(* CODESYS project Templates.export

Project tree, tasks and I/O mapping:
  Templates/
    Behaviour Model/
      function block ETrigATlTo_Temp [ST]: CleanupAction, CyclicAction, ExitAction, ResetAction, SampleAction, StartAction
      function block ETrigATl_Temp [ST]: CleanupAction, CyclicAction, ExitAction, ResetAction, SampleAction, StartAction
      function block ETrigATo_Temp [ST]: CleanupAction, CyclicAction, ExitAction, ResetAction, SampleAction, StartAction
      function block ETrigA_Temp [ST]: CleanupAction, CyclicAction, ExitAction, ResetAction, SampleAction, StartAction
      function block ETrigTlTo_Temp [ST]: CleanupAction, CyclicAction, ExitAction, ResetAction, SampleAction, StartAction
      function block ETrigTl_Temp [ST]: CleanupAction, CyclicAction, ExitAction, ResetAction, SampleAction, StartAction
      function block ETrigTo_Temp [ST]: CleanupAction, CyclicAction, ExitAction, ResetAction, SampleAction, StartAction
      function block ETrig_Temp [ST]: CleanupAction, CyclicAction, ExitAction, ResetAction, SampleAction, StartAction
      function block LConC_Temp [ST]: CleanupAction, CyclicAction, ExitAction, ResetAction, StartAction
      function block LConTlC_Temp [ST]: CleanupAction, CyclicAction, ExitAction, ResetAction, StartAction
      function block LConTlTo_Temp [ST]: CleanupAction, CyclicAction, ExitAction, ResetAction, StartAction
      function block LConTl_Temp [ST]: CleanupAction, CyclicAction, ExitAction, ResetAction, StartAction
      function block LConTo_Temp [ST]: CleanupAction, CyclicAction, ExitAction, ResetAction, StartAction
      function block LCon_Temp [ST]: CleanupAction, CyclicAction, ExitAction, ResetAction, StartAction
    FB Factory/
      function block CustomData [ST]
      function block CustomFB [ST]: prvInstInit
      function block CustomFBFactory_heap [ST]: Create, prvInstCount, prvInstPoolExtendsFactor, prvInstSize
      function block CustomFBFactory_static [ST]: Create, prvInstPoolAdr, prvInstPoolSize, prvInstSize
*)

// Templates/Behaviour Model/ETrigATlTo_Temp
//{attribute 'hide_all_locals'}
//{attribute 'conditionalshow_all_locals' := 'SomeText'}
//{attribute 'conditionalshow_all_locals'}
//{attribute 'conditionalshow' := 'SomeText'}
//{attribute 'conditionalshow'}
//{attribute 'hide'}
FUNCTION_BLOCK ETrigATlTo_Temp EXTENDS CBML.ETrigATlTo
VAR_INPUT
	(* specific Inputs *)
END_VAR
VAR_OUTPUT
	(* specific Outputs *)
	eErrorID : ERROR;
END_VAR
VAR
	(* specific vars *)
END_VAR

SUPER^();
IF _Model.iErrorID = CBML.ERROR.TIME_OUT THEN
	eErrorID := ERROR.TIME_OUT;
ELSE
	eErrorID := _Model.iErrorID;
END_IF

METHOD CleanupAction
VAR_INPUT
    xAbortProposed : BOOL;
    iErrorIDProposed: INT;
END_VAR
VAR_OUTPUT
    xComplete : BOOL := TRUE;
    xAbort: BOOL := xAbortProposed;
 	iErrorID : INT := iErrorIDProposed;
END_VAR
{analysis -2} 
/// ``CleanupAction`` is running until one of the following events occurs:
/// When ``xComplete`` is ``TRUE`` the state |STATE.DONE| is reached.
/// When ``xAbort`` is ``TRUE`` the state |STATE.ABORTED| is reached.
/// When ``iErrorID`` ≠ 0 (Zero) the state |STATE.ERROR| is reached.
///
/// | After a *Ready Condition* as input (``iErrorIDProposed`` = 0 and ``xAbortProposed`` = ``FALSE``), only the output states
/// | `DONE` (``xComplete`` is ``TRUE``) or `ERROR` (``iErrorID`` ≠ 0) are possible.
///
/// | After a *Error Condition* as input (``iErrorIDProposed`` ≠ 0), only the output state
/// | `ERROR` (``iErrorID`` ≠ 0) is possible.
///
/// | After a *Abort Condition* as Input (``xAbortProposed`` = ``TRUE``), only the output states
/// | `ABORTED` (``xAbort`` is ``TRUE``) or `ERROR` (``iErrorID`` ≠ 0) are possible.
///
/// .. admonition:: Example
///
///     .. code-block:: codesys
///     
///         (* common cleanup -- first steps *) 
///         
///         IF xComplete THEN
///             IF xAbortProposed THEN
///                 (* abort condition -- abort specific cleanup *)
///                 xAbort := TRUE;
///                 xComplete := FALSE;
///             ELSIF iErrorIDProposed <> 0 THEN
///                 (* error condition -- error specific cleanup *)
///                 iErrorID := SEL(xComplete, 0, iErrorIDProposed);
///                 xComplete := FALSE;
///             ELSE
///                 (* ready condition -- done specific cleanup*)
///             END_IF
///         END_IF
///
///         (* common cleanup -- last steps *) 
///
/// .. note::
///
///    If this method will not provide any implementation, please remove it!
END_METHOD

METHOD CyclicAction
VAR_INPUT
    itfTimingController : CBML.ITimingController;
END_VAR
VAR_OUTPUT
    xComplete : BOOL := TRUE;
    iErrorID : INT := 0;
END_VAR
{analysis -2} 
/// The CyclicAction is running until either ``xComplete`` is ``TRUE`` or ``iErrorID`` ≠  0 (Zero).
/// If ``xComplete`` is ``TRUE`` or ``iErrorID`` ≠  0 (Zero) the state |STATE.CLEANING| is reached.
/// With ``itfTimingController`` ≠  0 (Zero) it is possible to check the current invocation time (see: |ITimingController.ControllerCheckTiming|).
/// Function blocks with a ``udiTimeLimit`` input variable (see: |IETrigTl|, |IETrigATl|, |IETrigTlTo|, |IETrigATlTo|, |ILConTl|, |ILConTlTo|, |ILConTlC|)
/// should be implement in such a way that the current invocation is exited when the consumed time for this invocation has exceeded the settings from udiTimeLimit.
///
/// .. admonition:: Example
///
///     .. code-block:: codesys
///     
///         REPEAT
///             // working to reach the ready condition
///             // ⇒ xComplete := TRUE
///             // if the maximum invocation time is reached
///             // ⇒ xTimeLimit := TRUE
///             // if the maximum operating time is reached
///             // ⇒ xTimeOut := TRUE
///             // if an error condition is reached
///             // ⇒ set iErrorID to a value other than 0 (Zero)
///             itfTimingController.ControllerCheckTiming(
///                 xTimeOut=>xTimeOut,
///                 xTimeLimit=>xTimeLimit
///             );
///         
///             xComplete := TRUE;
///             iErrorID := ERROR.NO_ERROR;
///     
///         UNTIL xComplete OR
///               xTimeOut OR xTimeLimit OR
///               iErrorID <> ERROR.NO_ERROR
///         END_REPEAT
///
/// .. note::
///
///    If this method will not provide any implementation, please remove it!
END_METHOD

METHOD ExitAction
VAR_INPUT
    xAfterCleanup : BOOL;
    xInCopyCode : BOOL;
END_VAR
{analysis -2} 
/// This method is intended for releasing external resources (like RTS handles).
/// Do not call other internal function block instances in the context of this method.
/// Call only external functions defined inside the RTS.
/// For cleaning up other resources then external ones, please use the ``CleanupAction``.
/// This method should be callable in the context of ``FB_EXIT`` for example
/// before downloading a new application or before reseting an application.
///
/// .. note::
///
///    If this method will not provide any implementation, please remove it!
END_METHOD

METHOD ResetAction
VAR_OUTPUT
    xComplete : BOOL := TRUE;
END_VAR
{analysis -2} 
/// The ``ResetAction`` is running until the output ``xComplete`` is ``TRUE``.
/// If ``xComplete`` is ``TRUE`` the state |STATE.DORMANT| is reached.
///
/// .. note::
///
///    If this method will not provide any implementation, please remove it!
END_METHOD

METHOD SampleAction
VAR_OUTPUT
 	iErrorID : INT := 0;
END_VAR
{analysis -2} 
/// After leaving the state |STATE.DORMANT| the ``SampleAction`` is running one time then the state |STATE.STARTING| is reached.
/// If there is a ``iErrorID`` ≠  0 (Zero) the state |STATE.CLEANING| is reached instead.
///
/// .. note::
///
///    If this method will not provide any implementation, please remove it!
END_METHOD

METHOD StartAction
VAR_OUTPUT
    xComplete : BOOL := TRUE;
	iErrorID : INT := 0;
END_VAR
{analysis -2} 
/// The ``StartAction`` is running until either the output ``xComplete`` is ``TRUE`` or ``iErrorID`` ≠ 0 (Zero).
/// If ``xComplete`` is ``TRUE`` the state |STATE.EXECUTING| is reached.
/// If there is a ``iErrorID`` ≠  0 (Zero) the state |STATE.CLEANING| is reached.
///
/// .. note::
///
///    To sample the inputs in the first invocation of a function block the method SampleAction is the solution of choice.
///    See: |ISampleActionProvider.SampleAction|
///
/// .. note::
///
///    If this method will not provide any implementation, please remove it!
END_METHOD

END_FUNCTION_BLOCK

// Templates/Behaviour Model/ETrigATl_Temp
//{attribute 'hide_all_locals'}
//{attribute 'conditionalshow_all_locals' := 'SomeText'}
//{attribute 'conditionalshow_all_locals'}
//{attribute 'conditionalshow' := 'SomeText'}
//{attribute 'conditionalshow'}
//{attribute 'hide'}
FUNCTION_BLOCK ETrigATl_Temp EXTENDS CBML.ETrigATl
VAR_INPUT
	(* specific Inputs *)
END_VAR
VAR_OUTPUT
	eErrorID : ERROR;
	(* specific Outputs *)
END_VAR
VAR
	(* specific vars *)
END_VAR

SUPER^();
eErrorID := _Model.iErrorID;

METHOD CleanupAction
VAR_INPUT
    xAbortProposed : BOOL;
    iErrorIDProposed: INT;
END_VAR
VAR_OUTPUT
    xComplete : BOOL := TRUE;
    xAbort: BOOL := xAbortProposed;
 	iErrorID : INT := iErrorIDProposed;
END_VAR
{analysis -2} 
/// ``CleanupAction`` is running until one of the following events occurs:
/// When ``xComplete`` is ``TRUE`` the state |STATE.DONE| is reached.
/// When ``xAbort`` is ``TRUE`` the state |STATE.ABORTED| is reached.
/// When ``iErrorID`` ≠ 0 (Zero) the state |STATE.ERROR| is reached.
///
/// | After a *Ready Condition* as input (``iErrorIDProposed`` = 0 and ``xAbortProposed`` = ``FALSE``), only the output states
/// | `DONE` (``xComplete`` is ``TRUE``) or `ERROR` (``iErrorID`` ≠ 0) are possible.
///
/// | After a *Error Condition* as input (``iErrorIDProposed`` ≠ 0), only the output state
/// | `ERROR` (``iErrorID`` ≠ 0) is possible.
///
/// | After a *Abort Condition* as Input (``xAbortProposed`` = ``TRUE``), only the output states
/// | `ABORTED` (``xAbort`` is ``TRUE``) or `ERROR` (``iErrorID`` ≠ 0) are possible.
///
/// .. admonition:: Example
///
///     .. code-block:: codesys
///     
///         (* common cleanup -- first steps *) 
///         
///         IF xComplete THEN
///             IF xAbortProposed THEN
///                 (* abort condition -- abort specific cleanup *)
///                 xAbort := TRUE;
///                 xComplete := FALSE;
///             ELSIF iErrorIDProposed <> 0 THEN
///                 (* error condition -- error specific cleanup *)
///                 iErrorID := SEL(xComplete, 0, iErrorIDProposed);
///                 xComplete := FALSE;
///             ELSE
///                 (* ready condition -- done specific cleanup*)
///             END_IF
///         END_IF
///
///         (* common cleanup -- last steps *) 
///
/// .. note::
///
///    If this method will not provide any implementation, please remove it!
END_METHOD

METHOD CyclicAction
VAR_INPUT
    itfTimingController : CBML.ITimingController;
END_VAR
VAR_OUTPUT
    xComplete : BOOL := TRUE;
    iErrorID : INT := 0;
END_VAR
{analysis -2} 
/// The CyclicAction is running until either ``xComplete`` is ``TRUE`` or ``iErrorID`` ≠  0 (Zero).
/// If ``xComplete`` is ``TRUE`` or ``iErrorID`` ≠  0 (Zero) the state |STATE.CLEANING| is reached.
/// With ``itfTimingController`` ≠  0 (Zero) it is possible to check the current invocation time (see: |ITimingController.ControllerCheckTiming|).
/// Function blocks with a ``udiTimeLimit`` input variable (see: |IETrigTl|, |IETrigATl|, |IETrigTlTo|, |IETrigATlTo|, |ILConTl|, |ILConTlTo|, |ILConTlC|)
/// should be implement in such a way that the current invocation is exited when the consumed time for this invocation has exceeded the settings from udiTimeLimit.
///
/// .. admonition:: Example
///
///     .. code-block:: codesys
///     
///         REPEAT
///             // working to reach the ready condition
///             // ⇒ xComplete := TRUE
///             // if the maximum invocation time is reached
///             // ⇒ xTimeLimit := TRUE
///             // if the maximum operating time is reached
///             // ⇒ xTimeOut := TRUE
///             // if an error condition is reached
///             // ⇒ set iErrorID to a value other than 0 (Zero)
///             itfTimingController.ControllerCheckTiming(
///                 xTimeOut=>xTimeOut,
///                 xTimeLimit=>xTimeLimit
///             );
///         
///             xComplete := TRUE;
///             iErrorID := ERROR.NO_ERROR;
///     
///         UNTIL xComplete OR
///               xTimeOut OR xTimeLimit OR
///               iErrorID <> ERROR.NO_ERROR
///         END_REPEAT
///
/// .. note::
///
///    If this method will not provide any implementation, please remove it!
END_METHOD

METHOD ExitAction
VAR_INPUT
    xAfterCleanup : BOOL;
    xInCopyCode : BOOL;
END_VAR
{analysis -2} 
/// This method is intended for releasing external resources (like RTS handles).
/// Do not call other internal function block instances in the context of this method.
/// Call only external functions defined inside the RTS.
/// For cleaning up other resources then external ones, please use the ``CleanupAction``.
/// This method should be callable in the context of ``FB_EXIT`` for example
/// before downloading a new application or before reseting an application.
///
/// .. note::
///
///    If this method will not provide any implementation, please remove it!
END_METHOD

METHOD ResetAction
VAR_OUTPUT
    xComplete : BOOL := TRUE;
END_VAR
{analysis -2} 
/// The ``ResetAction`` is running until the output ``xComplete`` is ``TRUE``.
/// If ``xComplete`` is ``TRUE`` the state |STATE.DORMANT| is reached.
///
/// .. note::
///
///    If this method will not provide any implementation, please remove it!
END_METHOD

METHOD SampleAction
VAR_OUTPUT
 	iErrorID : INT := 0;
END_VAR
{analysis -2} 
/// After leaving the state |STATE.DORMANT| the ``SampleAction`` is running one time then the state |STATE.STARTING| is reached.
/// If there is a ``iErrorID`` ≠  0 (Zero) the state |STATE.CLEANING| is reached instead.
///
/// .. note::
///
///    If this method will not provide any implementation, please remove it!
END_METHOD

METHOD StartAction
VAR_OUTPUT
    xComplete : BOOL := TRUE;
	iErrorID : INT := 0;
END_VAR
{analysis -2} 
/// The ``StartAction`` is running until either the output ``xComplete`` is ``TRUE`` or ``iErrorID`` ≠ 0 (Zero).
/// If ``xComplete`` is ``TRUE`` the state |STATE.EXECUTING| is reached.
/// If there is a ``iErrorID`` ≠  0 (Zero) the state |STATE.CLEANING| is reached.
///
/// .. note::
///
///    To sample the inputs in the first invocation of a function block the method SampleAction is the solution of choice.
///    See: |ISampleActionProvider.SampleAction|
///
/// .. note::
///
///    If this method will not provide any implementation, please remove it!
END_METHOD

END_FUNCTION_BLOCK

// Templates/Behaviour Model/ETrigATo_Temp
//{attribute 'hide_all_locals'}
//{attribute 'conditionalshow_all_locals' := 'SomeText'}
//{attribute 'conditionalshow_all_locals'}
//{attribute 'conditionalshow' := 'SomeText'}
//{attribute 'conditionalshow'}
//{attribute 'hide'}
FUNCTION_BLOCK ETrigATo_Temp EXTENDS CBML.ETrigATo
VAR_INPUT
	(* specific Inputs *)
END_VAR
VAR_OUTPUT
	eErrorID : ERROR;
	(* specific Outputs *)
END_VAR
VAR
	(* specific vars *)
END_VAR

SUPER^();
IF _Model.iErrorID = CBML.ERROR.TIME_OUT THEN
	eErrorID := ERROR.TIME_OUT;
ELSE
	eErrorID := _Model.iErrorID;
END_IF

METHOD CleanupAction
VAR_INPUT
    xAbortProposed : BOOL;
    iErrorIDProposed: INT;
END_VAR
VAR_OUTPUT
    xComplete : BOOL := TRUE;
    xAbort: BOOL := xAbortProposed;
 	iErrorID : INT := iErrorIDProposed;
END_VAR
{analysis -2} 
/// ``CleanupAction`` is running until one of the following events occurs:
/// When ``xComplete`` is ``TRUE`` the state |STATE.DONE| is reached.
/// When ``xAbort`` is ``TRUE`` the state |STATE.ABORTED| is reached.
/// When ``iErrorID`` ≠ 0 (Zero) the state |STATE.ERROR| is reached.
///
/// | After a *Ready Condition* as input (``iErrorIDProposed`` = 0 and ``xAbortProposed`` = ``FALSE``), only the output states
/// | `DONE` (``xComplete`` is ``TRUE``) or `ERROR` (``iErrorID`` ≠ 0) are possible.
///
/// | After a *Error Condition* as input (``iErrorIDProposed`` ≠ 0), only the output state
/// | `ERROR` (``iErrorID`` ≠ 0) is possible.
///
/// | After a *Abort Condition* as Input (``xAbortProposed`` = ``TRUE``), only the output states
/// | `ABORTED` (``xAbort`` is ``TRUE``) or `ERROR` (``iErrorID`` ≠ 0) are possible.
///
/// .. admonition:: Example
///
///     .. code-block:: codesys
///     
///         (* common cleanup -- first steps *) 
///         
///         IF xComplete THEN
///             IF xAbortProposed THEN
///                 (* abort condition -- abort specific cleanup *)
///                 xAbort := TRUE;
///                 xComplete := FALSE;
///             ELSIF iErrorIDProposed <> 0 THEN
///                 (* error condition -- error specific cleanup *)
///                 iErrorID := SEL(xComplete, 0, iErrorIDProposed);
///                 xComplete := FALSE;
///             ELSE
///                 (* ready condition -- done specific cleanup*)
///             END_IF
///         END_IF
///
///         (* common cleanup -- last steps *) 
///
/// .. note::
///
///    If this method will not provide any implementation, please remove it!
END_METHOD

METHOD CyclicAction
VAR_INPUT
    itfTimingController : CBML.ITimingController;
END_VAR
VAR_OUTPUT
    xComplete : BOOL := TRUE;
    iErrorID : INT := 0;
END_VAR
{analysis -2} 
/// The CyclicAction is running until either ``xComplete`` is ``TRUE`` or ``iErrorID`` ≠  0 (Zero).
/// If ``xComplete`` is ``TRUE`` or ``iErrorID`` ≠  0 (Zero) the state |STATE.CLEANING| is reached.
/// With ``itfTimingController`` ≠  0 (Zero) it is possible to check the current invocation time (see: |ITimingController.ControllerCheckTiming|).
/// Function blocks with a ``udiTimeLimit`` input variable (see: |IETrigTl|, |IETrigATl|, |IETrigTlTo|, |IETrigATlTo|, |ILConTl|, |ILConTlTo|, |ILConTlC|)
/// should be implement in such a way that the current invocation is exited when the consumed time for this invocation has exceeded the settings from udiTimeLimit.
///
/// .. admonition:: Example
///
///     .. code-block:: codesys
///     
///         REPEAT
///             // working to reach the ready condition
///             // ⇒ xComplete := TRUE
///             // if the maximum invocation time is reached
///             // ⇒ xTimeLimit := TRUE
///             // if the maximum operating time is reached
///             // ⇒ xTimeOut := TRUE
///             // if an error condition is reached
///             // ⇒ set iErrorID to a value other than 0 (Zero)
///             itfTimingController.ControllerCheckTiming(
///                 xTimeOut=>xTimeOut,
///                 xTimeLimit=>xTimeLimit
///             );
///         
///             xComplete := TRUE;
///             iErrorID := ERROR.NO_ERROR;
///     
///         UNTIL xComplete OR
///               xTimeOut OR xTimeLimit OR
///               iErrorID <> ERROR.NO_ERROR
///         END_REPEAT
///
/// .. note::
///
///    If this method will not provide any implementation, please remove it!
END_METHOD

METHOD ExitAction
VAR_INPUT
    xAfterCleanup : BOOL;
    xInCopyCode : BOOL;
END_VAR
{analysis -2} 
/// This method is intended for releasing external resources (like RTS handles).
/// Do not call other internal function block instances in the context of this method.
/// Call only external functions defined inside the RTS.
/// For cleaning up other resources then external ones, please use the ``CleanupAction``.
/// This method should be callable in the context of ``FB_EXIT`` for example
/// before downloading a new application or before reseting an application.
///
/// .. note::
///
///    If this method will not provide any implementation, please remove it!
END_METHOD

METHOD ResetAction
VAR_OUTPUT
    xComplete : BOOL := TRUE;
END_VAR
{analysis -2} 
/// The ``ResetAction`` is running until the output ``xComplete`` is ``TRUE``.
/// If ``xComplete`` is ``TRUE`` the state |STATE.DORMANT| is reached.
///
/// .. note::
///
///    If this method will not provide any implementation, please remove it!
END_METHOD

METHOD SampleAction
VAR_OUTPUT
 	iErrorID : INT := 0;
END_VAR
{analysis -2} 
/// After leaving the state |STATE.DORMANT| the ``SampleAction`` is running one time then the state |STATE.STARTING| is reached.
/// If there is a ``iErrorID`` ≠  0 (Zero) the state |STATE.CLEANING| is reached instead.
///
/// .. note::
///
///    If this method will not provide any implementation, please remove it!
END_METHOD

METHOD StartAction
VAR_OUTPUT
    xComplete : BOOL := TRUE;
	iErrorID : INT := 0;
END_VAR
{analysis -2} 
/// The ``StartAction`` is running until either the output ``xComplete`` is ``TRUE`` or ``iErrorID`` ≠ 0 (Zero).
/// If ``xComplete`` is ``TRUE`` the state |STATE.EXECUTING| is reached.
/// If there is a ``iErrorID`` ≠  0 (Zero) the state |STATE.CLEANING| is reached.
///
/// .. note::
///
///    To sample the inputs in the first invocation of a function block the method SampleAction is the solution of choice.
///    See: |ISampleActionProvider.SampleAction|
///
/// .. note::
///
///    If this method will not provide any implementation, please remove it!
END_METHOD

END_FUNCTION_BLOCK

// Templates/Behaviour Model/ETrigA_Temp
//{attribute 'hide_all_locals'}
//{attribute 'conditionalshow_all_locals' := 'SomeText'}
//{attribute 'conditionalshow_all_locals'}
//{attribute 'conditionalshow' := 'SomeText'}
//{attribute 'conditionalshow'}
//{attribute 'hide'}
FUNCTION_BLOCK ETrigA_Temp EXTENDS CBML.ETrigA
VAR_INPUT
	(* specific Inputs *)
END_VAR
VAR_OUTPUT
	eErrorID : ERROR;
	(* specific Outputs *)
END_VAR
VAR
	(* specific vars *)
END_VAR

SUPER^();
eErrorID := _Model.iErrorID;

METHOD CleanupAction
VAR_INPUT
    xAbortProposed : BOOL;
    iErrorIDProposed: INT;
END_VAR
VAR_OUTPUT
    xComplete : BOOL := TRUE;
    xAbort: BOOL := xAbortProposed;
 	iErrorID : INT := iErrorIDProposed;
END_VAR
{analysis -2} 
/// ``CleanupAction`` is running until one of the following events occurs:
/// When ``xComplete`` is ``TRUE`` the state |STATE.DONE| is reached.
/// When ``xAbort`` is ``TRUE`` the state |STATE.ABORTED| is reached.
/// When ``iErrorID`` ≠ 0 (Zero) the state |STATE.ERROR| is reached.
///
/// | After a *Ready Condition* as input (``iErrorIDProposed`` = 0 and ``xAbortProposed`` = ``FALSE``), only the output states
/// | `DONE` (``xComplete`` is ``TRUE``) or `ERROR` (``iErrorID`` ≠ 0) are possible.
///
/// | After a *Error Condition* as input (``iErrorIDProposed`` ≠ 0), only the output state
/// | `ERROR` (``iErrorID`` ≠ 0) is possible.
///
/// | After a *Abort Condition* as Input (``xAbortProposed`` = ``TRUE``), only the output states
/// | `ABORTED` (``xAbort`` is ``TRUE``) or `ERROR` (``iErrorID`` ≠ 0) are possible.
///
/// .. admonition:: Example
///
///     .. code-block:: codesys
///     
///         (* common cleanup -- first steps *) 
///         
///         IF xComplete THEN
///             IF xAbortProposed THEN
///                 (* abort condition -- abort specific cleanup *)
///                 xAbort := TRUE;
///                 xComplete := FALSE;
///             ELSIF iErrorIDProposed <> 0 THEN
///                 (* error condition -- error specific cleanup *)
///                 iErrorID := SEL(xComplete, 0, iErrorIDProposed);
///                 xComplete := FALSE;
///             ELSE
///                 (* ready condition -- done specific cleanup*)
///             END_IF
///         END_IF
///
///         (* common cleanup -- last steps *) 
///
/// .. note::
///
///    If this method will not provide any implementation, please remove it!
END_METHOD

METHOD CyclicAction
VAR_INPUT
    itfTimingController : CBML.ITimingController;
END_VAR
VAR_OUTPUT
    xComplete : BOOL := TRUE;
    iErrorID : INT := 0;
END_VAR
{analysis -2} 
/// The CyclicAction is running until either ``xComplete`` is ``TRUE`` or ``iErrorID`` ≠  0 (Zero).
/// If ``xComplete`` is ``TRUE`` or ``iErrorID`` ≠  0 (Zero) the state |STATE.CLEANING| is reached.
/// With ``itfTimingController`` ≠  0 (Zero) it is possible to check the current invocation time (see: |ITimingController.ControllerCheckTiming|).
/// Function blocks with a ``udiTimeLimit`` input variable (see: |IETrigTl|, |IETrigATl|, |IETrigTlTo|, |IETrigATlTo|, |ILConTl|, |ILConTlTo|, |ILConTlC|)
/// should be implement in such a way that the current invocation is exited when the consumed time for this invocation has exceeded the settings from udiTimeLimit.
///
/// .. admonition:: Example
///
///     .. code-block:: codesys
///     
///         REPEAT
///             // working to reach the ready condition
///             // ⇒ xComplete := TRUE
///             // if the maximum invocation time is reached
///             // ⇒ xTimeLimit := TRUE
///             // if the maximum operating time is reached
///             // ⇒ xTimeOut := TRUE
///             // if an error condition is reached
///             // ⇒ set iErrorID to a value other than 0 (Zero)
///             itfTimingController.ControllerCheckTiming(
///                 xTimeOut=>xTimeOut,
///                 xTimeLimit=>xTimeLimit
///             );
///         
///             xComplete := TRUE;
///             iErrorID := ERROR.NO_ERROR;
///     
///         UNTIL xComplete OR
///               xTimeOut OR xTimeLimit OR
///               iErrorID <> ERROR.NO_ERROR
///         END_REPEAT
///
/// .. note::
///
///    If this method will not provide any implementation, please remove it!
END_METHOD

METHOD ExitAction
VAR_INPUT
    xAfterCleanup : BOOL;
    xInCopyCode : BOOL;
END_VAR
{analysis -2} 
/// This method is intended for releasing external resources (like RTS handles).
/// Do not call other internal function block instances in the context of this method.
/// Call only external functions defined inside the RTS.
/// For cleaning up other resources then external ones, please use the ``CleanupAction``.
/// This method should be callable in the context of ``FB_EXIT`` for example
/// before downloading a new application or before reseting an application.
///
/// .. note::
///
///    If this method will not provide any implementation, please remove it!
END_METHOD

METHOD ResetAction
VAR_OUTPUT
    xComplete : BOOL := TRUE;
END_VAR
{analysis -2} 
/// The ``ResetAction`` is running until the output ``xComplete`` is ``TRUE``.
/// If ``xComplete`` is ``TRUE`` the state |STATE.DORMANT| is reached.
///
/// .. note::
///
///    If this method will not provide any implementation, please remove it!
END_METHOD

METHOD SampleAction
VAR_OUTPUT
 	iErrorID : INT := 0;
END_VAR
{analysis -2} 
/// After leaving the state |STATE.DORMANT| the ``SampleAction`` is running one time then the state |STATE.STARTING| is reached.
/// If there is a ``iErrorID`` ≠  0 (Zero) the state |STATE.CLEANING| is reached instead.
///
/// .. note::
///
///    If this method will not provide any implementation, please remove it!
END_METHOD

METHOD StartAction
VAR_OUTPUT
    xComplete : BOOL := TRUE;
	iErrorID : INT := 0;
END_VAR
{analysis -2} 
/// The ``StartAction`` is running until either the output ``xComplete`` is ``TRUE`` or ``iErrorID`` ≠ 0 (Zero).
/// If ``xComplete`` is ``TRUE`` the state |STATE.EXECUTING| is reached.
/// If there is a ``iErrorID`` ≠  0 (Zero) the state |STATE.CLEANING| is reached.
///
/// .. note::
///
///    To sample the inputs in the first invocation of a function block the method SampleAction is the solution of choice.
///    See: |ISampleActionProvider.SampleAction|
///
/// .. note::
///
///    If this method will not provide any implementation, please remove it!
END_METHOD

END_FUNCTION_BLOCK

// Templates/Behaviour Model/ETrigTlTo_Temp
//{attribute 'hide_all_locals'}
//{attribute 'conditionalshow_all_locals' := 'SomeText'}
//{attribute 'conditionalshow_all_locals'}
//{attribute 'conditionalshow' := 'SomeText'}
//{attribute 'conditionalshow'}
//{attribute 'hide'}
FUNCTION_BLOCK ETrigTlTo_Temp EXTENDS CBML.ETrigTlTo
VAR_INPUT
	(* specific Inputs *)
END_VAR
VAR_OUTPUT
	eErrorID : ERROR;
	(* specific Outputs *)
END_VAR
VAR
	(* specific vars *)
END_VAR

SUPER^();
IF _Model.iErrorID = CBML.ERROR.TIME_OUT THEN
	eErrorID := ERROR.TIME_OUT;
ELSE
	eErrorID := _Model.iErrorID;
END_IF

METHOD CleanupAction
VAR_INPUT
    xAbortProposed : BOOL;
    iErrorIDProposed: INT;
END_VAR
VAR_OUTPUT
    xComplete : BOOL := TRUE;
    xAbort: BOOL := xAbortProposed;
 	iErrorID : INT := iErrorIDProposed;
END_VAR
{analysis -2} 
/// ``CleanupAction`` is running until one of the following events occurs:
/// When ``xComplete`` is ``TRUE`` the state |STATE.DONE| is reached.
/// When ``xAbort`` is ``TRUE`` the state |STATE.ABORTED| is reached.
/// When ``iErrorID`` ≠ 0 (Zero) the state |STATE.ERROR| is reached.
///
/// | After a *Ready Condition* as input (``iErrorIDProposed`` = 0 and ``xAbortProposed`` = ``FALSE``), only the output states
/// | `DONE` (``xComplete`` is ``TRUE``) or `ERROR` (``iErrorID`` ≠ 0) are possible.
///
/// | After a *Error Condition* as input (``iErrorIDProposed`` ≠ 0), only the output state
/// | `ERROR` (``iErrorID`` ≠ 0) is possible.
///
/// | After a *Abort Condition* as Input (``xAbortProposed`` = ``TRUE``), only the output states
/// | `ABORTED` (``xAbort`` is ``TRUE``) or `ERROR` (``iErrorID`` ≠ 0) are possible.
///
/// .. admonition:: Example
///
///     .. code-block:: codesys
///     
///         (* common cleanup -- first steps *) 
///         
///         IF xComplete THEN
///             IF xAbortProposed THEN
///                 (* abort condition -- abort specific cleanup *)
///                 xAbort := TRUE;
///                 xComplete := FALSE;
///             ELSIF iErrorIDProposed <> 0 THEN
///                 (* error condition -- error specific cleanup *)
///                 iErrorID := SEL(xComplete, 0, iErrorIDProposed);
///                 xComplete := FALSE;
///             ELSE
///                 (* ready condition -- done specific cleanup*)
///             END_IF
///         END_IF
///
///         (* common cleanup -- last steps *) 
///
/// .. note::
///
///    If this method will not provide any implementation, please remove it!
END_METHOD

METHOD CyclicAction
VAR_INPUT
    itfTimingController : CBML.ITimingController;
END_VAR
VAR_OUTPUT
    xComplete : BOOL := TRUE;
    iErrorID : INT := 0;
END_VAR
{analysis -2} 
/// The CyclicAction is running until either ``xComplete`` is ``TRUE`` or ``iErrorID`` ≠  0 (Zero).
/// If ``xComplete`` is ``TRUE`` or ``iErrorID`` ≠  0 (Zero) the state |STATE.CLEANING| is reached.
/// With ``itfTimingController`` ≠  0 (Zero) it is possible to check the current invocation time (see: |ITimingController.ControllerCheckTiming|).
/// Function blocks with a ``udiTimeLimit`` input variable (see: |IETrigTl|, |IETrigATl|, |IETrigTlTo|, |IETrigATlTo|, |ILConTl|, |ILConTlTo|, |ILConTlC|)
/// should be implement in such a way that the current invocation is exited when the consumed time for this invocation has exceeded the settings from udiTimeLimit.
///
/// .. admonition:: Example
///
///     .. code-block:: codesys
///     
///         REPEAT
///             // working to reach the ready condition
///             // ⇒ xComplete := TRUE
///             // if the maximum invocation time is reached
///             // ⇒ xTimeLimit := TRUE
///             // if the maximum operating time is reached
///             // ⇒ xTimeOut := TRUE
///             // if an error condition is reached
///             // ⇒ set iErrorID to a value other than 0 (Zero)
///             itfTimingController.ControllerCheckTiming(
///                 xTimeOut=>xTimeOut,
///                 xTimeLimit=>xTimeLimit
///             );
///         
///             xComplete := TRUE;
///             iErrorID := ERROR.NO_ERROR;
///     
///         UNTIL xComplete OR
///               xTimeOut OR xTimeLimit OR
///               iErrorID <> ERROR.NO_ERROR
///         END_REPEAT
///
/// .. note::
///
///    If this method will not provide any implementation, please remove it!
END_METHOD

METHOD ExitAction
VAR_INPUT
    xAfterCleanup : BOOL;
    xInCopyCode : BOOL;
END_VAR
{analysis -2} 
/// This method is intended for releasing external resources (like RTS handles).
/// Do not call other internal function block instances in the context of this method.
/// Call only external functions defined inside the RTS.
/// For cleaning up other resources then external ones, please use the ``CleanupAction``.
/// This method should be callable in the context of ``FB_EXIT`` for example
/// before downloading a new application or before reseting an application.
///
/// .. note::
///
///    If this method will not provide any implementation, please remove it!
END_METHOD

METHOD ResetAction
VAR_OUTPUT
    xComplete : BOOL := TRUE;
END_VAR
{analysis -2} 
/// The ``ResetAction`` is running until the output ``xComplete`` is ``TRUE``.
/// If ``xComplete`` is ``TRUE`` the state |STATE.DORMANT| is reached.
///
/// .. note::
///
///    If this method will not provide any implementation, please remove it!
END_METHOD

METHOD SampleAction
VAR_OUTPUT
 	iErrorID : INT := 0;
END_VAR
{analysis -2} 
/// After leaving the state |STATE.DORMANT| the ``SampleAction`` is running one time then the state |STATE.STARTING| is reached.
/// If there is a ``iErrorID`` ≠  0 (Zero) the state |STATE.CLEANING| is reached instead.
///
/// .. note::
///
///    If this method will not provide any implementation, please remove it!
END_METHOD

METHOD StartAction
VAR_OUTPUT
    xComplete : BOOL := TRUE;
	iErrorID : INT := 0;
END_VAR
{analysis -2} 
/// The ``StartAction`` is running until either the output ``xComplete`` is ``TRUE`` or ``iErrorID`` ≠ 0 (Zero).
/// If ``xComplete`` is ``TRUE`` the state |STATE.EXECUTING| is reached.
/// If there is a ``iErrorID`` ≠  0 (Zero) the state |STATE.CLEANING| is reached.
///
/// .. note::
///
///    To sample the inputs in the first invocation of a function block the method SampleAction is the solution of choice.
///    See: |ISampleActionProvider.SampleAction|
///
/// .. note::
///
///    If this method will not provide any implementation, please remove it!
END_METHOD

END_FUNCTION_BLOCK

// Templates/Behaviour Model/ETrigTl_Temp
//{attribute 'hide_all_locals'}
//{attribute 'conditionalshow_all_locals' := 'SomeText'}
//{attribute 'conditionalshow_all_locals'}
//{attribute 'conditionalshow' := 'SomeText'}
//{attribute 'conditionalshow'}
//{attribute 'hide'}
FUNCTION_BLOCK ETrigTl_Temp EXTENDS CBML.ETrigTl
VAR_INPUT
	(* specific Inputs *)
END_VAR
VAR_OUTPUT
	eErrorID : ERROR;
	(* specific Outputs *)
END_VAR
VAR
	(* specific vars *)
END_VAR

SUPER^();
eErrorID := _Model.iErrorID;

METHOD CleanupAction
VAR_INPUT
    xAbortProposed : BOOL;
    iErrorIDProposed: INT;
END_VAR
VAR_OUTPUT
    xComplete : BOOL := TRUE;
    xAbort: BOOL := xAbortProposed;
 	iErrorID : INT := iErrorIDProposed;
END_VAR
{analysis -2} 
/// ``CleanupAction`` is running until one of the following events occurs:
/// When ``xComplete`` is ``TRUE`` the state |STATE.DONE| is reached.
/// When ``xAbort`` is ``TRUE`` the state |STATE.ABORTED| is reached.
/// When ``iErrorID`` ≠ 0 (Zero) the state |STATE.ERROR| is reached.
///
/// | After a *Ready Condition* as input (``iErrorIDProposed`` = 0 and ``xAbortProposed`` = ``FALSE``), only the output states
/// | `DONE` (``xComplete`` is ``TRUE``) or `ERROR` (``iErrorID`` ≠ 0) are possible.
///
/// | After a *Error Condition* as input (``iErrorIDProposed`` ≠ 0), only the output state
/// | `ERROR` (``iErrorID`` ≠ 0) is possible.
///
/// | After a *Abort Condition* as Input (``xAbortProposed`` = ``TRUE``), only the output states
/// | `ABORTED` (``xAbort`` is ``TRUE``) or `ERROR` (``iErrorID`` ≠ 0) are possible.
///
/// .. admonition:: Example
///
///     .. code-block:: codesys
///     
///         (* common cleanup -- first steps *) 
///         
///         IF xComplete THEN
///             IF xAbortProposed THEN
///                 (* abort condition -- abort specific cleanup *)
///                 xAbort := TRUE;
///                 xComplete := FALSE;
///             ELSIF iErrorIDProposed <> 0 THEN
///                 (* error condition -- error specific cleanup *)
///                 iErrorID := SEL(xComplete, 0, iErrorIDProposed);
///                 xComplete := FALSE;
///             ELSE
///                 (* ready condition -- done specific cleanup*)
///             END_IF
///         END_IF
///
///         (* common cleanup -- last steps *) 
///
/// .. note::
///
///    If this method will not provide any implementation, please remove it!
END_METHOD

METHOD CyclicAction
VAR_INPUT
    itfTimingController : CBML.ITimingController;
END_VAR
VAR_OUTPUT
    xComplete : BOOL := TRUE;
    iErrorID : INT := 0;
END_VAR
{analysis -2} 
/// The CyclicAction is running until either ``xComplete`` is ``TRUE`` or ``iErrorID`` ≠  0 (Zero).
/// If ``xComplete`` is ``TRUE`` or ``iErrorID`` ≠  0 (Zero) the state |STATE.CLEANING| is reached.
/// With ``itfTimingController`` ≠  0 (Zero) it is possible to check the current invocation time (see: |ITimingController.ControllerCheckTiming|).
/// Function blocks with a ``udiTimeLimit`` input variable (see: |IETrigTl|, |IETrigATl|, |IETrigTlTo|, |IETrigATlTo|, |ILConTl|, |ILConTlTo|, |ILConTlC|)
/// should be implement in such a way that the current invocation is exited when the consumed time for this invocation has exceeded the settings from udiTimeLimit.
///
/// .. admonition:: Example
///
///     .. code-block:: codesys
///     
///         REPEAT
///             // working to reach the ready condition
///             // ⇒ xComplete := TRUE
///             // if the maximum invocation time is reached
///             // ⇒ xTimeLimit := TRUE
///             // if the maximum operating time is reached
///             // ⇒ xTimeOut := TRUE
///             // if an error condition is reached
///             // ⇒ set iErrorID to a value other than 0 (Zero)
///             itfTimingController.ControllerCheckTiming(
///                 xTimeOut=>xTimeOut,
///                 xTimeLimit=>xTimeLimit
///             );
///         
///             xComplete := TRUE;
///             iErrorID := ERROR.NO_ERROR;
///     
///         UNTIL xComplete OR
///               xTimeOut OR xTimeLimit OR
///               iErrorID <> ERROR.NO_ERROR
///         END_REPEAT
///
/// .. note::
///
///    If this method will not provide any implementation, please remove it!
END_METHOD

METHOD ExitAction
VAR_INPUT
    xAfterCleanup : BOOL;
    xInCopyCode : BOOL;
END_VAR
{analysis -2} 
/// This method is intended for releasing external resources (like RTS handles).
/// Do not call other internal function block instances in the context of this method.
/// Call only external functions defined inside the RTS.
/// For cleaning up other resources then external ones, please use the ``CleanupAction``.
/// This method should be callable in the context of ``FB_EXIT`` for example
/// before downloading a new application or before reseting an application.
///
/// .. note::
///
///    If this method will not provide any implementation, please remove it!
END_METHOD

METHOD ResetAction
VAR_OUTPUT
    xComplete : BOOL := TRUE;
END_VAR
{analysis -2} 
/// The ``ResetAction`` is running until the output ``xComplete`` is ``TRUE``.
/// If ``xComplete`` is ``TRUE`` the state |STATE.DORMANT| is reached.
///
/// .. note::
///
///    If this method will not provide any implementation, please remove it!
END_METHOD

METHOD SampleAction
VAR_OUTPUT
 	iErrorID : INT := 0;
END_VAR
{analysis -2} 
/// After leaving the state |STATE.DORMANT| the ``SampleAction`` is running one time then the state |STATE.STARTING| is reached.
/// If there is a ``iErrorID`` ≠  0 (Zero) the state |STATE.CLEANING| is reached instead.
///
/// .. note::
///
///    If this method will not provide any implementation, please remove it!
END_METHOD

METHOD StartAction
VAR_OUTPUT
    xComplete : BOOL := TRUE;
	iErrorID : INT := 0;
END_VAR
{analysis -2} 
/// The ``StartAction`` is running until either the output ``xComplete`` is ``TRUE`` or ``iErrorID`` ≠ 0 (Zero).
/// If ``xComplete`` is ``TRUE`` the state |STATE.EXECUTING| is reached.
/// If there is a ``iErrorID`` ≠  0 (Zero) the state |STATE.CLEANING| is reached.
///
/// .. note::
///
///    To sample the inputs in the first invocation of a function block the method SampleAction is the solution of choice.
///    See: |ISampleActionProvider.SampleAction|
///
/// .. note::
///
///    If this method will not provide any implementation, please remove it!
END_METHOD

END_FUNCTION_BLOCK

// Templates/Behaviour Model/ETrigTo_Temp
//{attribute 'hide_all_locals'}
//{attribute 'conditionalshow_all_locals' := 'SomeText'}
//{attribute 'conditionalshow_all_locals'}
//{attribute 'conditionalshow' := 'SomeText'}
//{attribute 'conditionalshow'}
//{attribute 'hide'}
FUNCTION_BLOCK ETrigTo_Temp EXTENDS CBML.ETrigTo
VAR_INPUT
	(* specific Inputs *)
END_VAR
VAR_OUTPUT
	eErrorID : ERROR;
	(* specific Outputs *)
END_VAR
VAR
	(* specific vars *)
END_VAR

SUPER^();
IF _Model.iErrorID = CBML.ERROR.TIME_OUT THEN
	eErrorID := ERROR.TIME_OUT;
ELSE
	eErrorID := _Model.iErrorID;
END_IF

METHOD CleanupAction
VAR_INPUT
    xAbortProposed : BOOL;
    iErrorIDProposed: INT;
END_VAR
VAR_OUTPUT
    xComplete : BOOL := TRUE;
    xAbort: BOOL := xAbortProposed;
 	iErrorID : INT := iErrorIDProposed;
END_VAR
{analysis -2} 
/// ``CleanupAction`` is running until one of the following events occurs:
/// When ``xComplete`` is ``TRUE`` the state |STATE.DONE| is reached.
/// When ``xAbort`` is ``TRUE`` the state |STATE.ABORTED| is reached.
/// When ``iErrorID`` ≠ 0 (Zero) the state |STATE.ERROR| is reached.
///
/// | After a *Ready Condition* as input (``iErrorIDProposed`` = 0 and ``xAbortProposed`` = ``FALSE``), only the output states
/// | `DONE` (``xComplete`` is ``TRUE``) or `ERROR` (``iErrorID`` ≠ 0) are possible.
///
/// | After a *Error Condition* as input (``iErrorIDProposed`` ≠ 0), only the output state
/// | `ERROR` (``iErrorID`` ≠ 0) is possible.
///
/// | After a *Abort Condition* as Input (``xAbortProposed`` = ``TRUE``), only the output states
/// | `ABORTED` (``xAbort`` is ``TRUE``) or `ERROR` (``iErrorID`` ≠ 0) are possible.
///
/// .. admonition:: Example
///
///     .. code-block:: codesys
///     
///         (* common cleanup -- first steps *) 
///         
///         IF xComplete THEN
///             IF xAbortProposed THEN
///                 (* abort condition -- abort specific cleanup *)
///                 xAbort := TRUE;
///                 xComplete := FALSE;
///             ELSIF iErrorIDProposed <> 0 THEN
///                 (* error condition -- error specific cleanup *)
///                 iErrorID := SEL(xComplete, 0, iErrorIDProposed);
///                 xComplete := FALSE;
///             ELSE
///                 (* ready condition -- done specific cleanup*)
///             END_IF
///         END_IF
///
///         (* common cleanup -- last steps *) 
///
/// .. note::
///
///    If this method will not provide any implementation, please remove it!
END_METHOD

METHOD CyclicAction
VAR_INPUT
    itfTimingController : CBML.ITimingController;
END_VAR
VAR_OUTPUT
    xComplete : BOOL := TRUE;
    iErrorID : INT := 0;
END_VAR
{analysis -2} 
/// The CyclicAction is running until either ``xComplete`` is ``TRUE`` or ``iErrorID`` ≠  0 (Zero).
/// If ``xComplete`` is ``TRUE`` or ``iErrorID`` ≠  0 (Zero) the state |STATE.CLEANING| is reached.
/// With ``itfTimingController`` ≠  0 (Zero) it is possible to check the current invocation time (see: |ITimingController.ControllerCheckTiming|).
/// Function blocks with a ``udiTimeLimit`` input variable (see: |IETrigTl|, |IETrigATl|, |IETrigTlTo|, |IETrigATlTo|, |ILConTl|, |ILConTlTo|, |ILConTlC|)
/// should be implement in such a way that the current invocation is exited when the consumed time for this invocation has exceeded the settings from udiTimeLimit.
///
/// .. admonition:: Example
///
///     .. code-block:: codesys
///     
///         REPEAT
///             // working to reach the ready condition
///             // ⇒ xComplete := TRUE
///             // if the maximum invocation time is reached
///             // ⇒ xTimeLimit := TRUE
///             // if the maximum operating time is reached
///             // ⇒ xTimeOut := TRUE
///             // if an error condition is reached
///             // ⇒ set iErrorID to a value other than 0 (Zero)
///             itfTimingController.ControllerCheckTiming(
///                 xTimeOut=>xTimeOut,
///                 xTimeLimit=>xTimeLimit
///             );
///         
///             xComplete := TRUE;
///             iErrorID := ERROR.NO_ERROR;
///     
///         UNTIL xComplete OR
///               xTimeOut OR xTimeLimit OR
///               iErrorID <> ERROR.NO_ERROR
///         END_REPEAT
///
/// .. note::
///
///    If this method will not provide any implementation, please remove it!
END_METHOD

METHOD ExitAction
VAR_INPUT
    xAfterCleanup : BOOL;
    xInCopyCode : BOOL;
END_VAR
{analysis -2} 
/// This method is intended for releasing external resources (like RTS handles).
/// Do not call other internal function block instances in the context of this method.
/// Call only external functions defined inside the RTS.
/// For cleaning up other resources then external ones, please use the ``CleanupAction``.
/// This method should be callable in the context of ``FB_EXIT`` for example
/// before downloading a new application or before reseting an application.
///
/// .. note::
///
///    If this method will not provide any implementation, please remove it!
END_METHOD

METHOD ResetAction
VAR_OUTPUT
    xComplete : BOOL := TRUE;
END_VAR
{analysis -2} 
/// The ``ResetAction`` is running until the output ``xComplete`` is ``TRUE``.
/// If ``xComplete`` is ``TRUE`` the state |STATE.DORMANT| is reached.
///
/// .. note::
///
///    If this method will not provide any implementation, please remove it!
END_METHOD

METHOD SampleAction
VAR_OUTPUT
 	iErrorID : INT := 0;
END_VAR
{analysis -2} 
/// After leaving the state |STATE.DORMANT| the ``SampleAction`` is running one time then the state |STATE.STARTING| is reached.
/// If there is a ``iErrorID`` ≠  0 (Zero) the state |STATE.CLEANING| is reached instead.
///
/// .. note::
///
///    If this method will not provide any implementation, please remove it!
END_METHOD

METHOD StartAction
VAR_OUTPUT
    xComplete : BOOL := TRUE;
	iErrorID : INT := 0;
END_VAR
{analysis -2} 
/// The ``StartAction`` is running until either the output ``xComplete`` is ``TRUE`` or ``iErrorID`` ≠ 0 (Zero).
/// If ``xComplete`` is ``TRUE`` the state |STATE.EXECUTING| is reached.
/// If there is a ``iErrorID`` ≠  0 (Zero) the state |STATE.CLEANING| is reached.
///
/// .. note::
///
///    To sample the inputs in the first invocation of a function block the method SampleAction is the solution of choice.
///    See: |ISampleActionProvider.SampleAction|
///
/// .. note::
///
///    If this method will not provide any implementation, please remove it!
END_METHOD

END_FUNCTION_BLOCK

// Templates/Behaviour Model/ETrig_Temp
//{attribute 'hide_all_locals'}
//{attribute 'conditionalshow_all_locals' := 'SomeText'}
//{attribute 'conditionalshow_all_locals'}
//{attribute 'conditionalshow' := 'SomeText'}
//{attribute 'conditionalshow'}
//{attribute 'hide'}
FUNCTION_BLOCK ETrig_Temp EXTENDS CBML.ETrig
VAR_INPUT
	(* specific Inputs *)
END_VAR
VAR_OUTPUT
	eErrorID : ERROR;
	(* specific Outputs *)
END_VAR
VAR
	(* specific vars *)
END_VAR

SUPER^();
eErrorID := _Model.iErrorID;

METHOD CleanupAction
VAR_INPUT
    xAbortProposed : BOOL;
    iErrorIDProposed: INT;
END_VAR
VAR_OUTPUT
    xComplete : BOOL := TRUE;
    xAbort: BOOL := xAbortProposed;
 	iErrorID : INT := iErrorIDProposed;
END_VAR
{analysis -2} 
/// ``CleanupAction`` is running until one of the following events occurs:
/// When ``xComplete`` is ``TRUE`` the state |STATE.DONE| is reached.
/// When ``xAbort`` is ``TRUE`` the state |STATE.ABORTED| is reached.
/// When ``iErrorID`` ≠ 0 (Zero) the state |STATE.ERROR| is reached.
///
/// | After a *Ready Condition* as input (``iErrorIDProposed`` = 0 and ``xAbortProposed`` = ``FALSE``), only the output states
/// | `DONE` (``xComplete`` is ``TRUE``) or `ERROR` (``iErrorID`` ≠ 0) are possible.
///
/// | After a *Error Condition* as input (``iErrorIDProposed`` ≠ 0), only the output state
/// | `ERROR` (``iErrorID`` ≠ 0) is possible.
///
/// | After a *Abort Condition* as Input (``xAbortProposed`` = ``TRUE``), only the output states
/// | `ABORTED` (``xAbort`` is ``TRUE``) or `ERROR` (``iErrorID`` ≠ 0) are possible.
///
/// .. admonition:: Example
///
///     .. code-block:: codesys
///     
///         (* common cleanup -- first steps *) 
///         
///         IF xComplete THEN
///             IF xAbortProposed THEN
///                 (* abort condition -- abort specific cleanup *)
///                 xAbort := TRUE;
///                 xComplete := FALSE;
///             ELSIF iErrorIDProposed <> 0 THEN
///                 (* error condition -- error specific cleanup *)
///                 iErrorID := SEL(xComplete, 0, iErrorIDProposed);
///                 xComplete := FALSE;
///             ELSE
///                 (* ready condition -- done specific cleanup*)
///             END_IF
///         END_IF
///
///         (* common cleanup -- last steps *) 
///
/// .. note::
///
///    If this method will not provide any implementation, please remove it!
END_METHOD

METHOD CyclicAction
VAR_INPUT
    itfTimingController : CBML.ITimingController;
END_VAR
VAR_OUTPUT
    xComplete : BOOL := TRUE;
    iErrorID : INT := 0;
END_VAR
{analysis -2} 
/// The CyclicAction is running until either ``xComplete`` is ``TRUE`` or ``iErrorID`` ≠  0 (Zero).
/// If ``xComplete`` is ``TRUE`` or ``iErrorID`` ≠  0 (Zero) the state |STATE.CLEANING| is reached.
/// With ``itfTimingController`` ≠  0 (Zero) it is possible to check the current invocation time (see: |ITimingController.ControllerCheckTiming|).
/// Function blocks with a ``udiTimeLimit`` input variable (see: |IETrigTl|, |IETrigATl|, |IETrigTlTo|, |IETrigATlTo|, |ILConTl|, |ILConTlTo|, |ILConTlC|)
/// should be implement in such a way that the current invocation is exited when the consumed time for this invocation has exceeded the settings from udiTimeLimit.
///
/// .. admonition:: Example
///
///     .. code-block:: codesys
///     
///         REPEAT
///             // working to reach the ready condition
///             // ⇒ xComplete := TRUE
///             // if the maximum invocation time is reached
///             // ⇒ xTimeLimit := TRUE
///             // if the maximum operating time is reached
///             // ⇒ xTimeOut := TRUE
///             // if an error condition is reached
///             // ⇒ set iErrorID to a value other than 0 (Zero)
///             itfTimingController.ControllerCheckTiming(
///                 xTimeOut=>xTimeOut,
///                 xTimeLimit=>xTimeLimit
///             );
///         
///             xComplete := TRUE;
///             iErrorID := ERROR.NO_ERROR;
///     
///         UNTIL xComplete OR
///               xTimeOut OR xTimeLimit OR
///               iErrorID <> ERROR.NO_ERROR
///         END_REPEAT
///
/// .. note::
///
///    If this method will not provide any implementation, please remove it!
END_METHOD

METHOD ExitAction
VAR_INPUT
    xAfterCleanup : BOOL;
    xInCopyCode : BOOL;
END_VAR
{analysis -2} 
/// This method is intended for releasing external resources (like RTS handles).
/// Do not call other internal function block instances in the context of this method.
/// Call only external functions defined inside the RTS.
/// For cleaning up other resources then external ones, please use the ``CleanupAction``.
/// This method should be callable in the context of ``FB_EXIT`` for example
/// before downloading a new application or before reseting an application.
///
/// .. note::
///
///    If this method will not provide any implementation, please remove it!
END_METHOD

METHOD ResetAction
VAR_OUTPUT
    xComplete : BOOL := TRUE;
END_VAR
{analysis -2} 
/// The ``ResetAction`` is running until the output ``xComplete`` is ``TRUE``.
/// If ``xComplete`` is ``TRUE`` the state |STATE.DORMANT| is reached.
///
/// .. note::
///
///    If this method will not provide any implementation, please remove it!
END_METHOD

METHOD SampleAction
VAR_OUTPUT
 	iErrorID : INT := 0;
END_VAR
{analysis -2} 
/// After leaving the state |STATE.DORMANT| the ``SampleAction`` is running one time then the state |STATE.STARTING| is reached.
/// If there is a ``iErrorID`` ≠  0 (Zero) the state |STATE.CLEANING| is reached instead.
///
/// .. note::
///
///    If this method will not provide any implementation, please remove it!
END_METHOD

METHOD StartAction
VAR_OUTPUT
    xComplete : BOOL := TRUE;
	iErrorID : INT := 0;
END_VAR
{analysis -2} 
/// The ``StartAction`` is running until either the output ``xComplete`` is ``TRUE`` or ``iErrorID`` ≠ 0 (Zero).
/// If ``xComplete`` is ``TRUE`` the state |STATE.EXECUTING| is reached.
/// If there is a ``iErrorID`` ≠  0 (Zero) the state |STATE.CLEANING| is reached.
///
/// .. note::
///
///    To sample the inputs in the first invocation of a function block the method SampleAction is the solution of choice.
///    See: |ISampleActionProvider.SampleAction|
///
/// .. note::
///
///    If this method will not provide any implementation, please remove it!
END_METHOD

END_FUNCTION_BLOCK

// Templates/Behaviour Model/LConC_Temp
//{attribute 'hide_all_locals'}
//{attribute 'conditionalshow_all_locals' := 'SomeText'}
//{attribute 'conditionalshow_all_locals'}
//{attribute 'conditionalshow' := 'SomeText'}
//{attribute 'conditionalshow'}
//{attribute 'hide'}
FUNCTION_BLOCK LConC_Temp EXTENDS CBML.LConC
VAR_INPUT
	(* specific Inputs *)
END_VAR
VAR_OUTPUT
	eErrorID : ERROR;
	(* specific Outputs *)
END_VAR
VAR
	(* specific vars *)
END_VAR

SUPER^();
eErrorID := _Model.iErrorID;

METHOD CleanupAction
VAR_INPUT
    xAbortProposed : BOOL;
    iErrorIDProposed: INT;
END_VAR
VAR_OUTPUT
    xComplete : BOOL := TRUE;
    xAbort: BOOL := xAbortProposed;
 	iErrorID : INT := iErrorIDProposed;
END_VAR
{analysis -2} 
/// ``CleanupAction`` is running until one of the following events occurs:
/// When ``xComplete`` is ``TRUE`` the state |STATE.DONE| is reached.
/// When ``xAbort`` is ``TRUE`` the state |STATE.ABORTED| is reached.
/// When ``iErrorID`` ≠ 0 (Zero) the state |STATE.ERROR| is reached.
///
/// | After a *Ready Condition* as input (``iErrorIDProposed`` = 0 and ``xAbortProposed`` = ``FALSE``), only the output states
/// | `DONE` (``xComplete`` is ``TRUE``) or `ERROR` (``iErrorID`` ≠ 0) are possible.
///
/// | After a *Error Condition* as input (``iErrorIDProposed`` ≠ 0), only the output state
/// | `ERROR` (``iErrorID`` ≠ 0) is possible.
///
/// | After a *Abort Condition* as Input (``xAbortProposed`` = ``TRUE``), only the output states
/// | `ABORTED` (``xAbort`` is ``TRUE``) or `ERROR` (``iErrorID`` ≠ 0) are possible.
///
/// .. admonition:: Example
///
///     .. code-block:: codesys
///     
///         (* common cleanup -- first steps *) 
///         
///         IF xComplete THEN
///             IF xAbortProposed THEN
///                 (* abort condition -- abort specific cleanup *)
///                 xAbort := TRUE;
///                 xComplete := FALSE;
///             ELSIF iErrorIDProposed <> 0 THEN
///                 (* error condition -- error specific cleanup *)
///                 iErrorID := SEL(xComplete, 0, iErrorIDProposed);
///                 xComplete := FALSE;
///             ELSE
///                 (* ready condition -- done specific cleanup*)
///             END_IF
///         END_IF
///
///         (* common cleanup -- last steps *) 
///
/// .. note::
///
///    If this method will not provide any implementation, please remove it!
END_METHOD

METHOD CyclicAction
VAR_INPUT
    itfTimingController : CBML.ITimingController;
END_VAR
VAR_OUTPUT
    xComplete : BOOL := TRUE;
    iErrorID : INT := 0;
END_VAR
{analysis -2} 
/// The CyclicAction is running until either ``xComplete`` is ``TRUE`` or ``iErrorID`` ≠  0 (Zero).
/// If ``xComplete`` is ``TRUE`` or ``iErrorID`` ≠  0 (Zero) the state |STATE.CLEANING| is reached.
/// With ``itfTimingController`` ≠  0 (Zero) it is possible to check the current invocation time (see: |ITimingController.ControllerCheckTiming|).
/// Function blocks with a ``udiTimeLimit`` input variable (see: |IETrigTl|, |IETrigATl|, |IETrigTlTo|, |IETrigATlTo|, |ILConTl|, |ILConTlTo|, |ILConTlC|)
/// should be implement in such a way that the current invocation is exited when the consumed time for this invocation has exceeded the settings from udiTimeLimit.
///
/// .. admonition:: Example
///
///     .. code-block:: codesys
///     
///         REPEAT
///             // working to reach the ready condition
///             // ⇒ xComplete := TRUE
///             // if the maximum invocation time is reached
///             // ⇒ xTimeLimit := TRUE
///             // if the maximum operating time is reached
///             // ⇒ xTimeOut := TRUE
///             // if an error condition is reached
///             // ⇒ set iErrorID to a value other than 0 (Zero)
///             itfTimingController.ControllerCheckTiming(
///                 xTimeOut=>xTimeOut,
///                 xTimeLimit=>xTimeLimit
///             );
///         
///             xComplete := TRUE;
///             iErrorID := ERROR.NO_ERROR;
///     
///         UNTIL xComplete OR
///               xTimeOut OR xTimeLimit OR
///               iErrorID <> ERROR.NO_ERROR
///         END_REPEAT
///
/// .. note::
///
///    If this method will not provide any implementation, please remove it!
END_METHOD

METHOD ExitAction
VAR_INPUT
    xAfterCleanup : BOOL;
    xInCopyCode : BOOL;
END_VAR
{analysis -2} 
/// This method is intended for releasing external resources (like RTS handles).
/// Do not call other internal function block instances in the context of this method.
/// Call only external functions defined inside the RTS.
/// For cleaning up other resources then external ones, please use the ``CleanupAction``.
/// This method should be callable in the context of ``FB_EXIT`` for example
/// before downloading a new application or before reseting an application.
///
/// .. note::
///
///    If this method will not provide any implementation, please remove it!
END_METHOD

METHOD ResetAction
VAR_OUTPUT
    xComplete : BOOL := TRUE;
END_VAR
{analysis -2} 
/// The ``ResetAction`` is running until the output ``xComplete`` is ``TRUE``.
/// If ``xComplete`` is ``TRUE`` the state |STATE.DORMANT| is reached.
///
/// .. note::
///
///    If this method will not provide any implementation, please remove it!
END_METHOD

METHOD StartAction
VAR_OUTPUT
    xComplete : BOOL := TRUE;
	iErrorID : INT := 0;
END_VAR
{analysis -2} 
/// The ``StartAction`` is running until either the output ``xComplete`` is ``TRUE`` or ``iErrorID`` ≠ 0 (Zero).
/// If ``xComplete`` is ``TRUE`` the state |STATE.EXECUTING| is reached.
/// If there is a ``iErrorID`` ≠  0 (Zero) the state |STATE.CLEANING| is reached.
///
/// .. note::
///
///    To sample the inputs in the first invocation of a function block the method SampleAction is the solution of choice.
///    See: |ISampleActionProvider.SampleAction|
///
/// .. note::
///
///    If this method will not provide any implementation, please remove it!
END_METHOD

END_FUNCTION_BLOCK

// Templates/Behaviour Model/LConTlC_Temp
//{attribute 'hide_all_locals'}
//{attribute 'conditionalshow_all_locals' := 'SomeText'}
//{attribute 'conditionalshow_all_locals'}
//{attribute 'conditionalshow' := 'SomeText'}
//{attribute 'conditionalshow'}
//{attribute 'hide'}
FUNCTION_BLOCK LConTlC_Temp EXTENDS CBML.LConTlC
VAR_INPUT
	(* specific Inputs *)
END_VAR
VAR_OUTPUT
	eErrorID : ERROR;
	(* specific Outputs *)
END_VAR
VAR
	(* specific vars *)
END_VAR

SUPER^();
eErrorID := _Model.iErrorID;

METHOD CleanupAction
VAR_INPUT
    xAbortProposed : BOOL;
    iErrorIDProposed: INT;
END_VAR
VAR_OUTPUT
    xComplete : BOOL := TRUE;
    xAbort: BOOL := xAbortProposed;
 	iErrorID : INT := iErrorIDProposed;
END_VAR
{analysis -2} 
/// ``CleanupAction`` is running until one of the following events occurs:
/// When ``xComplete`` is ``TRUE`` the state |STATE.DONE| is reached.
/// When ``xAbort`` is ``TRUE`` the state |STATE.ABORTED| is reached.
/// When ``iErrorID`` ≠ 0 (Zero) the state |STATE.ERROR| is reached.
///
/// | After a *Ready Condition* as input (``iErrorIDProposed`` = 0 and ``xAbortProposed`` = ``FALSE``), only the output states
/// | `DONE` (``xComplete`` is ``TRUE``) or `ERROR` (``iErrorID`` ≠ 0) are possible.
///
/// | After a *Error Condition* as input (``iErrorIDProposed`` ≠ 0), only the output state
/// | `ERROR` (``iErrorID`` ≠ 0) is possible.
///
/// | After a *Abort Condition* as Input (``xAbortProposed`` = ``TRUE``), only the output states
/// | `ABORTED` (``xAbort`` is ``TRUE``) or `ERROR` (``iErrorID`` ≠ 0) are possible.
///
/// .. admonition:: Example
///
///     .. code-block:: codesys
///     
///         (* common cleanup -- first steps *) 
///         
///         IF xComplete THEN
///             IF xAbortProposed THEN
///                 (* abort condition -- abort specific cleanup *)
///                 xAbort := TRUE;
///                 xComplete := FALSE;
///             ELSIF iErrorIDProposed <> 0 THEN
///                 (* error condition -- error specific cleanup *)
///                 iErrorID := SEL(xComplete, 0, iErrorIDProposed);
///                 xComplete := FALSE;
///             ELSE
///                 (* ready condition -- done specific cleanup*)
///             END_IF
///         END_IF
///
///         (* common cleanup -- last steps *) 
///
/// .. note::
///
///    If this method will not provide any implementation, please remove it!
END_METHOD

METHOD CyclicAction
VAR_INPUT
    itfTimingController : CBML.ITimingController;
END_VAR
VAR_OUTPUT
    xComplete : BOOL := TRUE;
    iErrorID : INT := 0;
END_VAR
{analysis -2} 
/// The CyclicAction is running until either ``xComplete`` is ``TRUE`` or ``iErrorID`` ≠  0 (Zero).
/// If ``xComplete`` is ``TRUE`` or ``iErrorID`` ≠  0 (Zero) the state |STATE.CLEANING| is reached.
/// With ``itfTimingController`` ≠  0 (Zero) it is possible to check the current invocation time (see: |ITimingController.ControllerCheckTiming|).
/// Function blocks with a ``udiTimeLimit`` input variable (see: |IETrigTl|, |IETrigATl|, |IETrigTlTo|, |IETrigATlTo|, |ILConTl|, |ILConTlTo|, |ILConTlC|)
/// should be implement in such a way that the current invocation is exited when the consumed time for this invocation has exceeded the settings from udiTimeLimit.
///
/// .. admonition:: Example
///
///     .. code-block:: codesys
///     
///         REPEAT
///             // working to reach the ready condition
///             // ⇒ xComplete := TRUE
///             // if the maximum invocation time is reached
///             // ⇒ xTimeLimit := TRUE
///             // if the maximum operating time is reached
///             // ⇒ xTimeOut := TRUE
///             // if an error condition is reached
///             // ⇒ set iErrorID to a value other than 0 (Zero)
///             itfTimingController.ControllerCheckTiming(
///                 xTimeOut=>xTimeOut,
///                 xTimeLimit=>xTimeLimit
///             );
///         
///             xComplete := TRUE;
///             iErrorID := ERROR.NO_ERROR;
///     
///         UNTIL xComplete OR
///               xTimeOut OR xTimeLimit OR
///               iErrorID <> ERROR.NO_ERROR
///         END_REPEAT
///
/// .. note::
///
///    If this method will not provide any implementation, please remove it!
END_METHOD

METHOD ExitAction
VAR_INPUT
    xAfterCleanup : BOOL;
    xInCopyCode : BOOL;
END_VAR
{analysis -2} 
/// This method is intended for releasing external resources (like RTS handles).
/// Do not call other internal function block instances in the context of this method.
/// Call only external functions defined inside the RTS.
/// For cleaning up other resources then external ones, please use the ``CleanupAction``.
/// This method should be callable in the context of ``FB_EXIT`` for example
/// before downloading a new application or before reseting an application.
///
/// .. note::
///
///    If this method will not provide any implementation, please remove it!
END_METHOD

METHOD ResetAction
VAR_OUTPUT
    xComplete : BOOL := TRUE;
END_VAR
{analysis -2} 
/// The ``ResetAction`` is running until the output ``xComplete`` is ``TRUE``.
/// If ``xComplete`` is ``TRUE`` the state |STATE.DORMANT| is reached.
///
/// .. note::
///
///    If this method will not provide any implementation, please remove it!
END_METHOD

METHOD StartAction
VAR_OUTPUT
    xComplete : BOOL := TRUE;
	iErrorID : INT := 0;
END_VAR
{analysis -2} 
/// The ``StartAction`` is running until either the output ``xComplete`` is ``TRUE`` or ``iErrorID`` ≠ 0 (Zero).
/// If ``xComplete`` is ``TRUE`` the state |STATE.EXECUTING| is reached.
/// If there is a ``iErrorID`` ≠  0 (Zero) the state |STATE.CLEANING| is reached.
///
/// .. note::
///
///    To sample the inputs in the first invocation of a function block the method SampleAction is the solution of choice.
///    See: |ISampleActionProvider.SampleAction|
///
/// .. note::
///
///    If this method will not provide any implementation, please remove it!
END_METHOD

END_FUNCTION_BLOCK

// Templates/Behaviour Model/LConTlTo_Temp
//{attribute 'hide_all_locals'}
//{attribute 'conditionalshow_all_locals' := 'SomeText'}
//{attribute 'conditionalshow_all_locals'}
//{attribute 'conditionalshow' := 'SomeText'}
//{attribute 'conditionalshow'}
//{attribute 'hide'}
FUNCTION_BLOCK LConTlTo_Temp EXTENDS CBML.LConTlTo
VAR_INPUT
	(* specific Inputs *)
END_VAR
VAR_OUTPUT
	eErrorID : ERROR;
	(* specific Outputs *)
END_VAR
VAR
	(* specific vars *)
END_VAR

SUPER^();
IF _Model.iErrorID = CBML.ERROR.TIME_OUT THEN
	eErrorID := ERROR.TIME_OUT;
ELSE
	eErrorID := _Model.iErrorID;
END_IF

METHOD CleanupAction
VAR_INPUT
    xAbortProposed : BOOL;
    iErrorIDProposed: INT;
END_VAR
VAR_OUTPUT
    xComplete : BOOL := TRUE;
    xAbort: BOOL := xAbortProposed;
 	iErrorID : INT := iErrorIDProposed;
END_VAR
{analysis -2} 
/// ``CleanupAction`` is running until one of the following events occurs:
/// When ``xComplete`` is ``TRUE`` the state |STATE.DONE| is reached.
/// When ``xAbort`` is ``TRUE`` the state |STATE.ABORTED| is reached.
/// When ``iErrorID`` ≠ 0 (Zero) the state |STATE.ERROR| is reached.
///
/// | After a *Ready Condition* as input (``iErrorIDProposed`` = 0 and ``xAbortProposed`` = ``FALSE``), only the output states
/// | `DONE` (``xComplete`` is ``TRUE``) or `ERROR` (``iErrorID`` ≠ 0) are possible.
///
/// | After a *Error Condition* as input (``iErrorIDProposed`` ≠ 0), only the output state
/// | `ERROR` (``iErrorID`` ≠ 0) is possible.
///
/// | After a *Abort Condition* as Input (``xAbortProposed`` = ``TRUE``), only the output states
/// | `ABORTED` (``xAbort`` is ``TRUE``) or `ERROR` (``iErrorID`` ≠ 0) are possible.
///
/// .. admonition:: Example
///
///     .. code-block:: codesys
///     
///         (* common cleanup -- first steps *) 
///         
///         IF xComplete THEN
///             IF xAbortProposed THEN
///                 (* abort condition -- abort specific cleanup *)
///                 xAbort := TRUE;
///                 xComplete := FALSE;
///             ELSIF iErrorIDProposed <> 0 THEN
///                 (* error condition -- error specific cleanup *)
///                 iErrorID := SEL(xComplete, 0, iErrorIDProposed);
///                 xComplete := FALSE;
///             ELSE
///                 (* ready condition -- done specific cleanup*)
///             END_IF
///         END_IF
///
///         (* common cleanup -- last steps *) 
///
/// .. note::
///
///    If this method will not provide any implementation, please remove it!
END_METHOD

METHOD CyclicAction
VAR_INPUT
    itfTimingController : CBML.ITimingController;
END_VAR
VAR_OUTPUT
    xComplete : BOOL := TRUE;
    iErrorID : INT := 0;
END_VAR
{analysis -2} 
/// The CyclicAction is running until either ``xComplete`` is ``TRUE`` or ``iErrorID`` ≠  0 (Zero).
/// If ``xComplete`` is ``TRUE`` or ``iErrorID`` ≠  0 (Zero) the state |STATE.CLEANING| is reached.
/// With ``itfTimingController`` ≠  0 (Zero) it is possible to check the current invocation time (see: |ITimingController.ControllerCheckTiming|).
/// Function blocks with a ``udiTimeLimit`` input variable (see: |IETrigTl|, |IETrigATl|, |IETrigTlTo|, |IETrigATlTo|, |ILConTl|, |ILConTlTo|, |ILConTlC|)
/// should be implement in such a way that the current invocation is exited when the consumed time for this invocation has exceeded the settings from udiTimeLimit.
///
/// .. admonition:: Example
///
///     .. code-block:: codesys
///     
///         REPEAT
///             // working to reach the ready condition
///             // ⇒ xComplete := TRUE
///             // if the maximum invocation time is reached
///             // ⇒ xTimeLimit := TRUE
///             // if the maximum operating time is reached
///             // ⇒ xTimeOut := TRUE
///             // if an error condition is reached
///             // ⇒ set iErrorID to a value other than 0 (Zero)
///             itfTimingController.ControllerCheckTiming(
///                 xTimeOut=>xTimeOut,
///                 xTimeLimit=>xTimeLimit
///             );
///         
///             xComplete := TRUE;
///             iErrorID := ERROR.NO_ERROR;
///     
///         UNTIL xComplete OR
///               xTimeOut OR xTimeLimit OR
///               iErrorID <> ERROR.NO_ERROR
///         END_REPEAT
///
/// .. note::
///
///    If this method will not provide any implementation, please remove it!
END_METHOD

METHOD ExitAction
VAR_INPUT
    xAfterCleanup : BOOL;
    xInCopyCode : BOOL;
END_VAR
{analysis -2} 
/// This method is intended for releasing external resources (like RTS handles).
/// Do not call other internal function block instances in the context of this method.
/// Call only external functions defined inside the RTS.
/// For cleaning up other resources then external ones, please use the ``CleanupAction``.
/// This method should be callable in the context of ``FB_EXIT`` for example
/// before downloading a new application or before reseting an application.
///
/// .. note::
///
///    If this method will not provide any implementation, please remove it!
END_METHOD

METHOD ResetAction
VAR_OUTPUT
    xComplete : BOOL := TRUE;
END_VAR
{analysis -2} 
/// The ``ResetAction`` is running until the output ``xComplete`` is ``TRUE``.
/// If ``xComplete`` is ``TRUE`` the state |STATE.DORMANT| is reached.
///
/// .. note::
///
///    If this method will not provide any implementation, please remove it!
END_METHOD

METHOD StartAction
VAR_OUTPUT
    xComplete : BOOL := TRUE;
	iErrorID : INT := 0;
END_VAR
{analysis -2} 
/// The ``StartAction`` is running until either the output ``xComplete`` is ``TRUE`` or ``iErrorID`` ≠ 0 (Zero).
/// If ``xComplete`` is ``TRUE`` the state |STATE.EXECUTING| is reached.
/// If there is a ``iErrorID`` ≠  0 (Zero) the state |STATE.CLEANING| is reached.
///
/// .. note::
///
///    To sample the inputs in the first invocation of a function block the method SampleAction is the solution of choice.
///    See: |ISampleActionProvider.SampleAction|
///
/// .. note::
///
///    If this method will not provide any implementation, please remove it!
END_METHOD

END_FUNCTION_BLOCK

// Templates/Behaviour Model/LConTl_Temp
//{attribute 'hide_all_locals'}
//{attribute 'conditionalshow_all_locals' := 'SomeText'}
//{attribute 'conditionalshow_all_locals'}
//{attribute 'conditionalshow' := 'SomeText'}
//{attribute 'conditionalshow'}
//{attribute 'hide'}
FUNCTION_BLOCK LConTl_Temp EXTENDS CBML.LConTl
VAR_INPUT
	(* specific Inputs *)
END_VAR
VAR_OUTPUT
	eErrorID : ERROR;
	(* specific Outputs *)
END_VAR
VAR
	(* specific vars *)
END_VAR

SUPER^();
eErrorID := _Model.iErrorID;

METHOD CleanupAction
VAR_INPUT
    xAbortProposed : BOOL;
    iErrorIDProposed: INT;
END_VAR
VAR_OUTPUT
    xComplete : BOOL := TRUE;
    xAbort: BOOL := xAbortProposed;
 	iErrorID : INT := iErrorIDProposed;
END_VAR
{analysis -2} 
/// ``CleanupAction`` is running until one of the following events occurs:
/// When ``xComplete`` is ``TRUE`` the state |STATE.DONE| is reached.
/// When ``xAbort`` is ``TRUE`` the state |STATE.ABORTED| is reached.
/// When ``iErrorID`` ≠ 0 (Zero) the state |STATE.ERROR| is reached.
///
/// | After a *Ready Condition* as input (``iErrorIDProposed`` = 0 and ``xAbortProposed`` = ``FALSE``), only the output states
/// | `DONE` (``xComplete`` is ``TRUE``) or `ERROR` (``iErrorID`` ≠ 0) are possible.
///
/// | After a *Error Condition* as input (``iErrorIDProposed`` ≠ 0), only the output state
/// | `ERROR` (``iErrorID`` ≠ 0) is possible.
///
/// | After a *Abort Condition* as Input (``xAbortProposed`` = ``TRUE``), only the output states
/// | `ABORTED` (``xAbort`` is ``TRUE``) or `ERROR` (``iErrorID`` ≠ 0) are possible.
///
/// .. admonition:: Example
///
///     .. code-block:: codesys
///     
///         (* common cleanup -- first steps *) 
///         
///         IF xComplete THEN
///             IF xAbortProposed THEN
///                 (* abort condition -- abort specific cleanup *)
///                 xAbort := TRUE;
///                 xComplete := FALSE;
///             ELSIF iErrorIDProposed <> 0 THEN
///                 (* error condition -- error specific cleanup *)
///                 iErrorID := SEL(xComplete, 0, iErrorIDProposed);
///                 xComplete := FALSE;
///             ELSE
///                 (* ready condition -- done specific cleanup*)
///             END_IF
///         END_IF
///
///         (* common cleanup -- last steps *) 
///
/// .. note::
///
///    If this method will not provide any implementation, please remove it!
END_METHOD

METHOD CyclicAction
VAR_INPUT
    itfTimingController : CBML.ITimingController;
END_VAR
VAR_OUTPUT
    xComplete : BOOL := TRUE;
    iErrorID : INT := 0;
END_VAR
{analysis -2} 
/// The CyclicAction is running until either ``xComplete`` is ``TRUE`` or ``iErrorID`` ≠  0 (Zero).
/// If ``xComplete`` is ``TRUE`` or ``iErrorID`` ≠  0 (Zero) the state |STATE.CLEANING| is reached.
/// With ``itfTimingController`` ≠  0 (Zero) it is possible to check the current invocation time (see: |ITimingController.ControllerCheckTiming|).
/// Function blocks with a ``udiTimeLimit`` input variable (see: |IETrigTl|, |IETrigATl|, |IETrigTlTo|, |IETrigATlTo|, |ILConTl|, |ILConTlTo|, |ILConTlC|)
/// should be implement in such a way that the current invocation is exited when the consumed time for this invocation has exceeded the settings from udiTimeLimit.
///
/// .. admonition:: Example
///
///     .. code-block:: codesys
///     
///         REPEAT
///             // working to reach the ready condition
///             // ⇒ xComplete := TRUE
///             // if the maximum invocation time is reached
///             // ⇒ xTimeLimit := TRUE
///             // if the maximum operating time is reached
///             // ⇒ xTimeOut := TRUE
///             // if an error condition is reached
///             // ⇒ set iErrorID to a value other than 0 (Zero)
///             itfTimingController.ControllerCheckTiming(
///                 xTimeOut=>xTimeOut,
///                 xTimeLimit=>xTimeLimit
///             );
///         
///             xComplete := TRUE;
///             iErrorID := ERROR.NO_ERROR;
///     
///         UNTIL xComplete OR
///               xTimeOut OR xTimeLimit OR
///               iErrorID <> ERROR.NO_ERROR
///         END_REPEAT
///
/// .. note::
///
///    If this method will not provide any implementation, please remove it!
END_METHOD

METHOD ExitAction
VAR_INPUT
    xAfterCleanup : BOOL;
    xInCopyCode : BOOL;
END_VAR
{analysis -2} 
/// This method is intended for releasing external resources (like RTS handles).
/// Do not call other internal function block instances in the context of this method.
/// Call only external functions defined inside the RTS.
/// For cleaning up other resources then external ones, please use the ``CleanupAction``.
/// This method should be callable in the context of ``FB_EXIT`` for example
/// before downloading a new application or before reseting an application.
///
/// .. note::
///
///    If this method will not provide any implementation, please remove it!
END_METHOD

METHOD ResetAction
VAR_OUTPUT
    xComplete : BOOL := TRUE;
END_VAR
{analysis -2} 
/// The ``ResetAction`` is running until the output ``xComplete`` is ``TRUE``.
/// If ``xComplete`` is ``TRUE`` the state |STATE.DORMANT| is reached.
///
/// .. note::
///
///    If this method will not provide any implementation, please remove it!
END_METHOD

METHOD StartAction
VAR_OUTPUT
    xComplete : BOOL := TRUE;
	iErrorID : INT := 0;
END_VAR
{analysis -2} 
/// The ``StartAction`` is running until either the output ``xComplete`` is ``TRUE`` or ``iErrorID`` ≠ 0 (Zero).
/// If ``xComplete`` is ``TRUE`` the state |STATE.EXECUTING| is reached.
/// If there is a ``iErrorID`` ≠  0 (Zero) the state |STATE.CLEANING| is reached.
///
/// .. note::
///
///    To sample the inputs in the first invocation of a function block the method SampleAction is the solution of choice.
///    See: |ISampleActionProvider.SampleAction|
///
/// .. note::
///
///    If this method will not provide any implementation, please remove it!
END_METHOD

END_FUNCTION_BLOCK

// Templates/Behaviour Model/LConTo_Temp
//{attribute 'hide_all_locals'}
//{attribute 'conditionalshow_all_locals' := 'SomeText'}
//{attribute 'conditionalshow_all_locals'}
//{attribute 'conditionalshow' := 'SomeText'}
//{attribute 'conditionalshow'}
//{attribute 'hide'}
FUNCTION_BLOCK LConTo_Temp EXTENDS CBML.LConTo
VAR_INPUT
	(* specific Inputs *)
END_VAR
VAR_OUTPUT
	eErrorID : ERROR;
	(* specific Outputs *)
END_VAR
VAR
	(* specific vars *)
END_VAR

SUPER^();
IF _Model.iErrorID = CBML.ERROR.TIME_OUT THEN
	eErrorID := ERROR.TIME_OUT;
ELSE
	eErrorID := _Model.iErrorID;
END_IF

METHOD CleanupAction
VAR_INPUT
    xAbortProposed : BOOL;
    iErrorIDProposed: INT;
END_VAR
VAR_OUTPUT
    xComplete : BOOL := TRUE;
    xAbort: BOOL := xAbortProposed;
 	iErrorID : INT := iErrorIDProposed;
END_VAR
{analysis -2} 
/// ``CleanupAction`` is running until one of the following events occurs:
/// When ``xComplete`` is ``TRUE`` the state |STATE.DONE| is reached.
/// When ``xAbort`` is ``TRUE`` the state |STATE.ABORTED| is reached.
/// When ``iErrorID`` ≠ 0 (Zero) the state |STATE.ERROR| is reached.
///
/// | After a *Ready Condition* as input (``iErrorIDProposed`` = 0 and ``xAbortProposed`` = ``FALSE``), only the output states
/// | `DONE` (``xComplete`` is ``TRUE``) or `ERROR` (``iErrorID`` ≠ 0) are possible.
///
/// | After a *Error Condition* as input (``iErrorIDProposed`` ≠ 0), only the output state
/// | `ERROR` (``iErrorID`` ≠ 0) is possible.
///
/// | After a *Abort Condition* as Input (``xAbortProposed`` = ``TRUE``), only the output states
/// | `ABORTED` (``xAbort`` is ``TRUE``) or `ERROR` (``iErrorID`` ≠ 0) are possible.
///
/// .. admonition:: Example
///
///     .. code-block:: codesys
///     
///         (* common cleanup -- first steps *) 
///         
///         IF xComplete THEN
///             IF xAbortProposed THEN
///                 (* abort condition -- abort specific cleanup *)
///                 xAbort := TRUE;
///                 xComplete := FALSE;
///             ELSIF iErrorIDProposed <> 0 THEN
///                 (* error condition -- error specific cleanup *)
///                 iErrorID := SEL(xComplete, 0, iErrorIDProposed);
///                 xComplete := FALSE;
///             ELSE
///                 (* ready condition -- done specific cleanup*)
///             END_IF
///         END_IF
///
///         (* common cleanup -- last steps *) 
///
/// .. note::
///
///    If this method will not provide any implementation, please remove it!
END_METHOD

METHOD CyclicAction
VAR_INPUT
    itfTimingController : CBML.ITimingController;
END_VAR
VAR_OUTPUT
    xComplete : BOOL := TRUE;
    iErrorID : INT := 0;
END_VAR
{analysis -2} 
/// The CyclicAction is running until either ``xComplete`` is ``TRUE`` or ``iErrorID`` ≠  0 (Zero).
/// If ``xComplete`` is ``TRUE`` or ``iErrorID`` ≠  0 (Zero) the state |STATE.CLEANING| is reached.
/// With ``itfTimingController`` ≠  0 (Zero) it is possible to check the current invocation time (see: |ITimingController.ControllerCheckTiming|).
/// Function blocks with a ``udiTimeLimit`` input variable (see: |IETrigTl|, |IETrigATl|, |IETrigTlTo|, |IETrigATlTo|, |ILConTl|, |ILConTlTo|, |ILConTlC|)
/// should be implement in such a way that the current invocation is exited when the consumed time for this invocation has exceeded the settings from udiTimeLimit.
///
/// .. admonition:: Example
///
///     .. code-block:: codesys
///     
///         REPEAT
///             // working to reach the ready condition
///             // ⇒ xComplete := TRUE
///             // if the maximum invocation time is reached
///             // ⇒ xTimeLimit := TRUE
///             // if the maximum operating time is reached
///             // ⇒ xTimeOut := TRUE
///             // if an error condition is reached
///             // ⇒ set iErrorID to a value other than 0 (Zero)
///             itfTimingController.ControllerCheckTiming(
///                 xTimeOut=>xTimeOut,
///                 xTimeLimit=>xTimeLimit
///             );
///         
///             xComplete := TRUE;
///             iErrorID := ERROR.NO_ERROR;
///     
///         UNTIL xComplete OR
///               xTimeOut OR xTimeLimit OR
///               iErrorID <> ERROR.NO_ERROR
///         END_REPEAT
///
/// .. note::
///
///    If this method will not provide any implementation, please remove it!
END_METHOD

METHOD ExitAction
VAR_INPUT
    xAfterCleanup : BOOL;
    xInCopyCode : BOOL;
END_VAR
{analysis -2} 
/// This method is intended for releasing external resources (like RTS handles).
/// Do not call other internal function block instances in the context of this method.
/// Call only external functions defined inside the RTS.
/// For cleaning up other resources then external ones, please use the ``CleanupAction``.
/// This method should be callable in the context of ``FB_EXIT`` for example
/// before downloading a new application or before reseting an application.
///
/// .. note::
///
///    If this method will not provide any implementation, please remove it!
END_METHOD

METHOD ResetAction
VAR_OUTPUT
    xComplete : BOOL := TRUE;
END_VAR
{analysis -2} 
/// The ``ResetAction`` is running until the output ``xComplete`` is ``TRUE``.
/// If ``xComplete`` is ``TRUE`` the state |STATE.DORMANT| is reached.
///
/// .. note::
///
///    If this method will not provide any implementation, please remove it!
END_METHOD

METHOD StartAction
VAR_OUTPUT
    xComplete : BOOL := TRUE;
	iErrorID : INT := 0;
END_VAR
{analysis -2} 
/// The ``StartAction`` is running until either the output ``xComplete`` is ``TRUE`` or ``iErrorID`` ≠ 0 (Zero).
/// If ``xComplete`` is ``TRUE`` the state |STATE.EXECUTING| is reached.
/// If there is a ``iErrorID`` ≠  0 (Zero) the state |STATE.CLEANING| is reached.
///
/// .. note::
///
///    To sample the inputs in the first invocation of a function block the method SampleAction is the solution of choice.
///    See: |ISampleActionProvider.SampleAction|
///
/// .. note::
///
///    If this method will not provide any implementation, please remove it!
END_METHOD

END_FUNCTION_BLOCK

// Templates/Behaviour Model/LCon_Temp
//{attribute 'hide_all_locals'}
//{attribute 'conditionalshow_all_locals' := 'SomeText'}
//{attribute 'conditionalshow_all_locals'}
//{attribute 'conditionalshow' := 'SomeText'}
//{attribute 'conditionalshow'}
//{attribute 'hide'}
FUNCTION_BLOCK LCon_Temp EXTENDS CBML.LCon
VAR_INPUT
	(* specific Inputs *)
END_VAR
VAR_OUTPUT
	eErrorID : ERROR;
	(* specific Outputs *)
END_VAR
VAR
	(* specific vars *)
END_VAR

SUPER^();
eErrorID := _Model.iErrorID;

METHOD CleanupAction
VAR_INPUT
    xAbortProposed : BOOL;
    iErrorIDProposed: INT;
END_VAR
VAR_OUTPUT
    xComplete : BOOL := TRUE;
    xAbort: BOOL := xAbortProposed;
 	iErrorID : INT := iErrorIDProposed;
END_VAR
{analysis -2} 
/// ``CleanupAction`` is running until one of the following events occurs:
/// When ``xComplete`` is ``TRUE`` the state |STATE.DONE| is reached.
/// When ``xAbort`` is ``TRUE`` the state |STATE.ABORTED| is reached.
/// When ``iErrorID`` ≠ 0 (Zero) the state |STATE.ERROR| is reached.
///
/// | After a *Ready Condition* as input (``iErrorIDProposed`` = 0 and ``xAbortProposed`` = ``FALSE``), only the output states
/// | `DONE` (``xComplete`` is ``TRUE``) or `ERROR` (``iErrorID`` ≠ 0) are possible.
///
/// | After a *Error Condition* as input (``iErrorIDProposed`` ≠ 0), only the output state
/// | `ERROR` (``iErrorID`` ≠ 0) is possible.
///
/// | After a *Abort Condition* as Input (``xAbortProposed`` = ``TRUE``), only the output states
/// | `ABORTED` (``xAbort`` is ``TRUE``) or `ERROR` (``iErrorID`` ≠ 0) are possible.
///
/// .. admonition:: Example
///
///     .. code-block:: codesys
///     
///         (* common cleanup -- first steps *) 
///         
///         IF xComplete THEN
///             IF xAbortProposed THEN
///                 (* abort condition -- abort specific cleanup *)
///                 xAbort := TRUE;
///                 xComplete := FALSE;
///             ELSIF iErrorIDProposed <> 0 THEN
///                 (* error condition -- error specific cleanup *)
///                 iErrorID := SEL(xComplete, 0, iErrorIDProposed);
///                 xComplete := FALSE;
///             ELSE
///                 (* ready condition -- done specific cleanup*)
///             END_IF
///         END_IF
///
///         (* common cleanup -- last steps *) 
///
/// .. note::
///
///    If this method will not provide any implementation, please remove it!
END_METHOD

METHOD CyclicAction
VAR_INPUT
    itfTimingController : CBML.ITimingController;
END_VAR
VAR_OUTPUT
    xComplete : BOOL := TRUE;
    iErrorID : INT := 0;
END_VAR
{analysis -2} 
/// The CyclicAction is running until either ``xComplete`` is ``TRUE`` or ``iErrorID`` ≠  0 (Zero).
/// If ``xComplete`` is ``TRUE`` or ``iErrorID`` ≠  0 (Zero) the state |STATE.CLEANING| is reached.
/// With ``itfTimingController`` ≠  0 (Zero) it is possible to check the current invocation time (see: |ITimingController.ControllerCheckTiming|).
/// Function blocks with a ``udiTimeLimit`` input variable (see: |IETrigTl|, |IETrigATl|, |IETrigTlTo|, |IETrigATlTo|, |ILConTl|, |ILConTlTo|, |ILConTlC|)
/// should be implement in such a way that the current invocation is exited when the consumed time for this invocation has exceeded the settings from udiTimeLimit.
///
/// .. admonition:: Example
///
///     .. code-block:: codesys
///     
///         REPEAT
///             // working to reach the ready condition
///             // ⇒ xComplete := TRUE
///             // if the maximum invocation time is reached
///             // ⇒ xTimeLimit := TRUE
///             // if the maximum operating time is reached
///             // ⇒ xTimeOut := TRUE
///             // if an error condition is reached
///             // ⇒ set iErrorID to a value other than 0 (Zero)
///             itfTimingController.ControllerCheckTiming(
///                 xTimeOut=>xTimeOut,
///                 xTimeLimit=>xTimeLimit
///             );
///         
///             xComplete := TRUE;
///             iErrorID := ERROR.NO_ERROR;
///     
///         UNTIL xComplete OR
///               xTimeOut OR xTimeLimit OR
///               iErrorID <> ERROR.NO_ERROR
///         END_REPEAT
///
/// .. note::
///
///    If this method will not provide any implementation, please remove it!
END_METHOD

METHOD ExitAction
VAR_INPUT
    xAfterCleanup : BOOL;
    xInCopyCode : BOOL;
END_VAR
{analysis -2} 
/// This method is intended for releasing external resources (like RTS handles).
/// Do not call other internal function block instances in the context of this method.
/// Call only external functions defined inside the RTS.
/// For cleaning up other resources then external ones, please use the ``CleanupAction``.
/// This method should be callable in the context of ``FB_EXIT`` for example
/// before downloading a new application or before reseting an application.
///
/// .. note::
///
///    If this method will not provide any implementation, please remove it!
END_METHOD

METHOD ResetAction
VAR_OUTPUT
    xComplete : BOOL := TRUE;
END_VAR
{analysis -2} 
/// The ``ResetAction`` is running until the output ``xComplete`` is ``TRUE``.
/// If ``xComplete`` is ``TRUE`` the state |STATE.DORMANT| is reached.
///
/// .. note::
///
///    If this method will not provide any implementation, please remove it!
END_METHOD

METHOD StartAction
VAR_OUTPUT
    xComplete : BOOL := TRUE;
	iErrorID : INT := 0;
END_VAR
{analysis -2} 
/// The ``StartAction`` is running until either the output ``xComplete`` is ``TRUE`` or ``iErrorID`` ≠ 0 (Zero).
/// If ``xComplete`` is ``TRUE`` the state |STATE.EXECUTING| is reached.
/// If there is a ``iErrorID`` ≠  0 (Zero) the state |STATE.CLEANING| is reached.
///
/// .. note::
///
///    To sample the inputs in the first invocation of a function block the method SampleAction is the solution of choice.
///    See: |ISampleActionProvider.SampleAction|
///
/// .. note::
///
///    If this method will not provide any implementation, please remove it!
END_METHOD

END_FUNCTION_BLOCK

// Templates/FB Factory/CustomData
// This is a container to carry init data from the Create methode of the factory
// to the prvInstInit methode of the new generated function block instance
{attribute 'enable_dynamic_creation'}
//{attribute 'hide_all_locals'}
//{attribute 'conditionalshow_all_locals' := 'SomeText'}
//{attribute 'conditionalshow_all_locals'}
//{attribute 'conditionalshow' := 'SomeText'}
//{attribute 'conditionalshow'}
//{attribute 'hide'}
FUNCTION_BLOCK CustomData EXTENDS FBF.InstanceData
VAR_INPUT
	(* Todo: Add your application specific data as input variables *)
END_VAR

(* !! Do not add any executable code here !! *)
SUPER^();

END_FUNCTION_BLOCK

// Templates/FB Factory/CustomFB
{attribute 'enable_dynamic_creation'}
//{attribute 'hide_all_locals'}
//{attribute 'conditionalshow_all_locals' := 'SomeText'}
//{attribute 'conditionalshow_all_locals'}
//{attribute 'conditionalshow' := 'SomeText'}
//{attribute 'conditionalshow'}
//{attribute 'hide'}
FUNCTION_BLOCK CustomFB EXTENDS FBF.InstanceBase;
VAR_INPUT
END_VAR
VAR_OUTPUT
END_VAR
VAR
END_VAR

SUPER^();

// This methode is called from the factory to give a chance
// to initialize the new fb instance with the content of itfData
//{attribute 'hide_all_locals'}
//{attribute 'conditionalshow_all_locals' := 'SomeText'}
//{attribute 'conditionalshow_all_locals'}
//{attribute 'conditionalshow' := 'SomeText'}
//{attribute 'conditionalshow'}
//{attribute 'hide'}
METHOD prvInstInit : FBF.ERROR
VAR_INPUT
	itfData : FBF.IData; 
END_VAR
VAR
	pData : POINTER TO CustomData;
	xOk : BOOL;
END_VAR
SUPER^.prvInstInit(itfData);
xOk := __QUERYPOINTER(itfData, pData);
IF xOk THEN
	(* THIS^.iLocalVar := pData^.iInitValue *);
END_IF
END_METHOD

END_FUNCTION_BLOCK

// Templates/FB Factory/CustomFBFactory_heap
// This is a template for a factory with an heap based extendable memory pool
{attribute 'enable_dynamic_creation'}
//{attribute 'hide_all_locals'}
//{attribute 'conditionalshow_all_locals' := 'SomeText'}
//{attribute 'conditionalshow_all_locals'}
//{attribute 'conditionalshow' := 'SomeText'}
//{attribute 'conditionalshow'}
//{attribute 'hide'}
FUNCTION_BLOCK CustomFBFactory_heap EXTENDS FBF.FactoryBase
VAR
END_VAR

SUPER^();

(* Please replace CustonFB with your specific function block type *)
(* There is no need to change anything else !!! *)
METHOD Create : POINTER TO CustomFB
VAR_INPUT
	itfData : FBF.IData;
END_VAR
VAR_OUTPUT
	eError : FBF.ERROR;
END_VAR
VAR
	hInst : CAA.HANDLE;
	itfInst : FBF.IInstance;
	xOk : BOOL;
END_VAR
(* !!! This code must not be subject to change !!! *)
hInst := SUPER^.prvAllocInstMem(eError => eError);
Create := SUPER^.prvGetInstPointer(hInst);
IF Create <> 0 AND eError = FBF.ERROR.NO_ERROR THEN

	{implicit on}
	Create^.__vfInit();
	Create^.FB_Init(TRUE, FALSE);
	{implicit off}

	xOk := __QUERYINTERFACE(Create^, itfInst);
	IF xOk THEN
		xOk := SUPER^.prvInstInit(itfInst, hInst, itfData, eError=>eError);
	ELSE
		eError := FBF.ERROR.WRONG_INTERFACE;
	END_IF

	IF NOT xOk THEN
		SUPER^.prvFreeInstMem(hInst);
		Create := CAA.gc_pNULL;
	END_IF
END_IF
END_METHOD

//{attribute 'conditionalshow' := 'SomeText'}
//{attribute 'conditionalshow'}
//{attribute 'hide'}
PROPERTY prvInstCount : CAA.COUNT (* ctInst *)
GET
(* Please choose a proper value for prvInstCount *)
prvInstCount := 10;
END_GET
END_PROPERTY

//{attribute 'conditionalshow' := 'SomeText'}
//{attribute 'conditionalshow'}
//{attribute 'hide'}
PROPERTY prvInstPoolExtendsFactor : USINT (* usiFactor [0..x%] *)
GET
(* Please choose a proper value for prvInstPoolExtendsFactor *)
(* This value will be interpreted as a 0..x% size extendsion related to the original size of the pool *)
prvInstPoolExtendsFactor := 20;
END_GET
END_PROPERTY

//{attribute 'conditionalshow' := 'SomeText'}
//{attribute 'conditionalshow'}
//{attribute 'hide'}
PROPERTY prvInstSize : CAA.SIZE (* szInst *)
GET
(* Please replace CustomFB with your specific function block type *)
prvInstSize := sizeof(CustomFB);
END_GET
END_PROPERTY

END_FUNCTION_BLOCK

// Templates/FB Factory/CustomFBFactory_static
// This is a template for a factory with an static iec memory based memory pool which a fixed capacity
{attribute 'enable_dynamic_creation'}
//{attribute 'hide_all_locals'}
//{attribute 'conditionalshow_all_locals' := 'SomeText'}
//{attribute 'conditionalshow_all_locals'}
//{attribute 'conditionalshow' := 'SomeText'}
//{attribute 'conditionalshow'}
//{attribute 'hide'}
FUNCTION_BLOCK CustomFBFactory_static EXTENDS FBF.FactoryBase
VAR
	// Please change the size of abyPoolMemory with your specific application need
	abyPoolMemory : ARRAY[0..529] OF BYTE;
END_VAR

SUPER^();

(* Please replace CustonFB with our specific function block type *)
(* There is no need to change anything else !!! *)
METHOD Create : POINTER TO CustomFB
VAR_INPUT
	itfData : FBF.IData;
END_VAR
VAR_OUTPUT
	eError : FBF.ERROR;
END_VAR
VAR
	hInst : CAA.HANDLE;
	itfInst : FBF.IInstance;
	xOk : BOOL;
END_VAR
(* !!! This code must not be subject to change !!! *)
hInst := SUPER^.prvAllocInstMem(eError => eError);
Create := SUPER^.prvGetInstPointer(hInst);
IF Create <> 0 AND eError = FBF.ERROR.NO_ERROR THEN

	{implicit on}
	Create^.__vfInit();
	Create^.FB_Init(TRUE, FALSE);
	{implicit off}

	xOk := __QUERYINTERFACE(Create^, itfInst);
	IF xOk THEN
		xOk := SUPER^.prvInstInit(itfInst, hInst, itfData, eError=>eError);
	ELSE
		eError := FBF.ERROR.WRONG_INTERFACE;
	END_IF

	IF NOT xOk THEN
		SUPER^.prvFreeInstMem(hInst);
		Create := CAA.gc_pNULL;
	END_IF
END_IF
END_METHOD

//{attribute 'conditionalshow' := 'SomeText'}
//{attribute 'conditionalshow'}
//{attribute 'hide'}
PROPERTY prvInstPoolAdr : CAA.PVOID (* pPool *)
GET
prvInstPoolAdr := ADR(abyPoolMemory);
END_GET
END_PROPERTY

//{attribute 'conditionalshow' := 'SomeText'}
//{attribute 'conditionalshow'}
//{attribute 'hide'}
PROPERTY prvInstPoolSize : CAA.SIZE (* szPool *)
GET
prvInstPoolSize := sizeof(abyPoolMemory);
END_GET
END_PROPERTY

//{attribute 'conditionalshow' := 'SomeText'}
//{attribute 'conditionalshow'}
//{attribute 'hide'}
PROPERTY prvInstSize : CAA.SIZE (* szInst *)
GET
(* Please replace CustomFB with your specific function block type *)
prvInstSize := sizeof(CustomFB);
END_GET
END_PROPERTY

END_FUNCTION_BLOCK
